	// cycle through coord system
	IF OptionsRtrig.Q AND NOT Controller.P_State.Buttons.Share THEN
		CASE _SMC_GroupJog2.CoordSystem OF
			SMC_COORD_SYSTEM.ACS:
				_SMC_GroupJog2.CoordSystem := SMC_COORD_SYSTEM.MCS;
				Controller.M_SetPlayerID(E_ControllerPlayerID.Player2);
			SMC_COORD_SYSTEM.MCS:
				_SMC_GroupJog2.CoordSystem := SMC_COORD_SYSTEM.PCS_1;
				Controller.M_SetPlayerID(E_ControllerPlayerID.Player3);
			SMC_COORD_SYSTEM.PCS_1:
				_SMC_GroupJog2.CoordSystem := SMC_COORD_SYSTEM.PCS_2;
				Controller.M_SetPlayerID(E_ControllerPlayerID.Player4);
			SMC_COORD_SYSTEM.PCS_2:
				_SMC_GroupJog2.CoordSystem := SMC_COORD_SYSTEM.TCS;
				Controller.M_SetPlayerID(E_ControllerPlayerID.PlayerALL);
			SMC_COORD_SYSTEM.TCS:
				_SMC_GroupJog2.CoordSystem := SMC_COORD_SYSTEM.ACS; // skip WCS
				Controller.M_SetPlayerID(E_ControllerPlayerID.Player1);
			SMC_COORD_SYSTEM.WCS:
				_SMC_GroupJog2.CoordSystem := SMC_COORD_SYSTEM.ACS;
				Controller.M_SetPlayerID(E_ControllerPlayerID.Player1);
		END_CASE
	END_IF
	
	// toggle the ABC as ACS setting
	IF ShareRtrig.Q AND NOT Controller.P_State.Buttons.Options THEN
		_SMC_GroupJog2.ABC_as_ACS := NOT _SMC_GroupJog2.ABC_as_ACS;
	END_IF
	
	// set the velocity factor while the left trigger button is pressed
	IF Controller.P_State.Dpad.Left AND_THEN Controller.P_State.Triggers.Right.Two <> R2_Last THEN
		R2_Last := Controller.P_State.Triggers.Right.Two;
		_SMC_GroupJog2.VelFactor := MAX(FactorMin, Controller.P_State.Triggers.Right.Two * 1.0 / 255.0);
	END_IF
	// set the acceleration factor while the up dpad button is pressed
	IF Controller.P_State.Dpad.Up AND_THEN Controller.P_State.Triggers.Right.Two <> R2_Last THEN
		R2_Last := Controller.P_State.Triggers.Right.Two;
		_SMC_GroupJog2.AccFactor := MAX(FactorMin, Controller.P_State.Triggers.Right.Two * 1.0 / 255.0);
	END_IF
	// set the jerk factor while the right dpad button is pressed
	IF Controller.P_State.Dpad.Right AND_THEN Controller.P_State.Triggers.Right.Two <> R2_Last THEN
		R2_Last := Controller.P_State.Triggers.Right.Two;
		_SMC_GroupJog2.JerkFactor := MAX(FactorMin, Controller.P_State.Triggers.Right.Two * 1.0 / 255.0);
	END_IF
	// set the torque factor while the down dpad down is pressed
	IF Controller.P_State.Dpad.Down AND_THEN Controller.P_State.Triggers.Right.Two <> R2_Last THEN
		R2_Last := Controller.P_State.Triggers.Right.Two;
		_SMC_GroupJog2.TorqueFactor := MAX(FactorMin, Controller.P_State.Triggers.Right.Two * 1.0 / 255.0);
	END_IF
	
	// first 4 poses can be called using buttons
	SquareButtonRtrig(CLK:=Controller.P_State.Buttons.Square);
	IF SquareButtonRtrig.Q THEN
		M_MoveToPose(E_Pose.One);
	END_IF
	TriangleButtonRtrig(CLK:=Controller.P_State.Buttons.Triangle);
	IF TriangleButtonRtrig.Q THEN
		M_MoveToPose(E_Pose.Two);
	END_IF
	CircleButtonRtrig(CLK:=Controller.P_State.Buttons.Circle);
	IF CircleButtonRtrig.Q THEN
		M_MoveToPose(E_Pose.Three);
	END_IF
	CrossButtonRtrig(CLK:=Controller.P_State.Buttons.Cross);
	IF CrossButtonRtrig.Q THEN
		M_MoveToPose(E_Pose.Four);
	END_IF
	
	//
	IF _SequenceMain = STEP_WAIT_JOG THEN
		
		//
		IF Controller.P_State.Joysticks.Left.X <> JoyStickLeftXLast
			OR Controller.P_State.Joysticks.Left.Y <> JoyStickLeftYLast THEN
				//
				JoyStickLeftXLast := Controller.P_State.Joysticks.Left.X;
				JoyStickLeftYLast := Controller.P_State.Joysticks.Left.Y;
				//	
				IF NOT Controller.P_State.Triggers.Left.One THEN
					// disable
					_SMC_GroupJog2.Forward[0] := FALSE;
					// disable
					_SMC_GroupJog2.Backward[0] := FALSE;
					// Controller.P_State.Joysticks.Left.X // X0-128 is -Y (Backward[1])
					_SMC_GroupJog2.Backward[1] := Controller.P_State.Joysticks.Left.X < _ControllerCenter - _ControllerDeadZone;
					// Controller.P_State.Joysticks.Left.X // X128-256 is +Y (Forward[1])
					_SMC_GroupJog2.Forward[1] := Controller.P_State.Joysticks.Left.X > _ControllerCenter + _ControllerDeadZone;
					// Controller.P_State.Joysticks.Left.Y // Y0-128 is +Z (Forward[2])
					_SMC_GroupJog2.Forward[2] := Controller.P_State.Joysticks.Left.Y < _ControllerCenter - _ControllerDeadZone;
					// Controller.P_State.Joysticks.Left.Y // Y128-256 is -Z (Backward[2])
					_SMC_GroupJog2.Backward[2] := Controller.P_State.Joysticks.Left.Y > _ControllerCenter + _ControllerDeadZone;
				ELSE
					// Controller.P_State.Joysticks.Left.Y // Y0-128 is +X (Forward[0])
					_SMC_GroupJog2.Forward[0] := Controller.P_State.Joysticks.Left.Y < _ControllerCenter - _ControllerDeadZone;
					// Controller.P_State.Joysticks.Left.Y // Y128-256 is -X (Backward[0])
					_SMC_GroupJog2.Backward[0] := Controller.P_State.Joysticks.Left.Y > _ControllerCenter + _ControllerDeadZone;
					// disable
					_SMC_GroupJog2.Backward[1] := FALSE;
					// disable
					_SMC_GroupJog2.Forward[1] := FALSE;
					// disable
					_SMC_GroupJog2.Forward[2] := FALSE;
					// disable])
					_SMC_GroupJog2.Backward[2] := FALSE;
				END_IF
		END_IF

		//
		IF Controller.P_State.Joysticks.Right.X <> JoyStickRightXLast
			OR Controller.P_State.Joysticks.Right.Y <> JoyStickRightYLast THEN
				//
				JoyStickRightXLast := Controller.P_State.Joysticks.Right.X;
				JoyStickRightYLast := Controller.P_State.Joysticks.Right.Y;
				//				
				IF NOT Controller.P_State.Triggers.Right.One THEN
					// Controller.P_State.Joysticks.Right.X // X0-128 is +Roll (rot about x) (Forward[3])
					_SMC_GroupJog2.Backward[3] := Controller.P_State.Joysticks.Right.X > _ControllerCenter + _ControllerDeadZone;
					// Controller.P_State.Joysticks.Right.X // X128-256 is -Roll (rot about x) (Backward[3])
					_SMC_GroupJog2.Forward[3] := Controller.P_State.Joysticks.Right.X < _ControllerCenter - _ControllerDeadZone;
					// Controller.P_State.Joysticks.Right.Y // Y0-128 is +Pitch (rot about y) (Forward[4])
					_SMC_GroupJog2.Forward[4] := Controller.P_State.Joysticks.Right.Y < _ControllerCenter - _ControllerDeadZone;
					// Controller.P_State.Joysticks.Right.Y // Y128-256 is -Pitch (rot about y) (Backward[4])
					_SMC_GroupJog2.Backward[4] := Controller.P_State.Joysticks.Right.Y > _ControllerCenter + _ControllerDeadZone;
					// disable
					_SMC_GroupJog2.Backward[5] := FALSE;
					// disable
					_SMC_GroupJog2.Forward[5] := FALSE;
				ELSE
					// disable
					_SMC_GroupJog2.Backward[3] := FALSE;
					// disable
					_SMC_GroupJog2.Forward[3] := FALSE;
					// disable
					_SMC_GroupJog2.Forward[4] := FALSE;
					// disable
					_SMC_GroupJog2.Backward[4] := FALSE;
					// Controller.P_State.Joysticks.Right.X // X0-128 is -Yaw (rot about z) (Backward[5])
					_SMC_GroupJog2.Backward[5] := Controller.P_State.Joysticks.Right.X < _ControllerCenter - _ControllerDeadZone;
					// Controller.P_State.Joysticks.Right.X // X128-256 is +Yaw (rot about z) (Forward[5])
					_SMC_GroupJog2.Forward[5] := Controller.P_State.Joysticks.Right.X > _ControllerCenter + _ControllerDeadZone;
				END_IF
		END_IF

	END_IF
	
END_IF
                        
END_METHOD

METHOD PRIVATE _M_CheckOffsets : BOOL
VAR_INPUT
END_VAR
VAR
	_i, _j, _k: INT;
END_VAR
                          IF _SMC_GroupJog2.Enable THEN
	FOR _j:=0 TO GVL.MCS_POS_IDX-GVL.TCP_POS_IDX BY 1 DO
		_OffsetExist[_j] := FALSE;
	END_FOR
	FOR _i := GVL.TCP_POS_IDX TO GVL.MCS_POS_IDX BY 1 DO
		IF StoredPositions[_i].Position.X <> 0
			OR_ELSE StoredPositions[_i].Position.Y <> 0
			OR_ELSE StoredPositions[_i].Position.Z <> 0
			OR_ELSE StoredPositions[_i].Position.A <> 0
			OR_ELSE StoredPositions[_i].Position.B <> 0
			OR_ELSE StoredPositions[_i].Position.C <> 0 THEN
				_OffsetExist[_i - GVL.TCP_POS_IDX] := TRUE;
		END_IF
	END_FOR
END_IF
                        
END_METHOD

METHOD PUBLIC M_ClearOffsets : BOOL
VAR_INPUT
END_VAR
                          
FOR _j:=0 TO 3 BY 1 DO
	_OffsetExist[_j] := FALSE;
END_FOR
FOR _i := GVL.TCP_POS_IDX TO GVL.MCS_POS_IDX BY 1 DO
	StoredPositions[_i].Position.X := 0.0;
	StoredPositions[_i].Position.Y := 0.0;
	StoredPositions[_i].Position.Z := 0.0;
	StoredPositions[_i].Position.A := 0.0;
	StoredPositions[_i].Position.B := 0.0;
	StoredPositions[_i].Position.C := 0.0;
END_FOR
                        
END_METHOD

METHOD PRIVATE _M_HandlePose : BOOL
VAR_IN_OUT
	AxisGroup: AXIS_GROUP_REF_SM3;
	GroupHandler: FB_GroupHandler;
END_VAR
VAR_INPUT
END_VAR
VAR
	_MoveCommand: ST_MoveCmd;
	_PoseSpeed: LREAL:=20.0;
END_VAR
                          FOR _i:=0 TO GVL.POSE_5_IDX - GVL.POSE_1_IDX BY 1 DO
	IF _MoveToPose[_i] THEN
		_MoveToPose[_i] := FALSE;
		//
		IF GVL.Enable 
			AND_THEN PersistentVars.Flags[GVL.HOME_COMPLETE].Value
			AND_THEN NOT _MoveCommandProcessor.Busy
			AND_THEN NOT _MoveCommandProcessor.Error THEN
				//
				_MoveCommand.MoveType 			:= DUT_Command_MoveType.DirectMove;
				_MoveCommand.PositionType 		:= DUT_Command_PositionType.AbsolutePosition;
				_MoveCommand.CoordinateType 	:= DUT_Command_CoordinateType.Literal;
				_MoveCommand.Speed 				:= _PoseSpeed;
				_MoveCommand.CoordSystem 		:= SMC_COORD_SYSTEM.ACS;
				_MoveCommand.CoordRef 			:= PersistentVars.StoredPositions[GVL.POSE_1_IDX + _i].Position;
				//
				_MoveCommandProcessor.Command := F_BuildMoveCmd(_MoveCommand);
				_MoveCommandProcessor.M_Start();
				//
				EXIT;
		END_IF;
	END_IF
END_FOR

_MoveCommandProcessor(
	StoredPositions:= StoredPositions,
	VisionRegisters:= VisionRegisters,
	Flags:= Flags,
	AxisGroup:= AxisGroup, 
	GroupHandler:= GroupHandler,
	Velocity:= StoredPositions[GVL.SPEEDS_IDX].Position.X, 
	VelFactor:= StoredPositions[GVL.SPEEDS_IDX].Position.A,
	Acceleration:= StoredPositions[GVL.SPEEDS_IDX].Position.Y, 
	AccFactor:= StoredPositions[GVL.SPEEDS_IDX].Position.B,
	Jerk:= StoredPositions[GVL.SPEEDS_IDX].Position.Z,
	JerkFactor:= StoredPositions[GVL.SPEEDS_IDX].Position.C, 
	Position=> ,
	ItfUnitMode=> , 
	Error=> );
                        
END_METHOD

METHOD PUBLIC M_MoveToPose : BOOL
VAR_INPUT
	Pose: E_Pose;
END_VAR
                          IF Enabled 
	AND NOT _MoveCommandProcessor.Busy
	AND NOT _MoveCommandProcessor.Error THEN
		M_MoveToPose := TRUE;
		_MoveToPose[Pose] := TRUE;
ELSE
	M_MoveToPose := FALSE;
END_IF
                        
END_METHOD
END_FUNCTION_BLOCK

FUNCTION_BLOCK FB_CommandProcessor EXTENDS FB_Module
VAR_IN_OUT
	J1, J2, J3, J4, J5, J6: AXIS_REF_SM3;
	AxisGroup: AXIS_GROUP_REF_SM3;
	GroupHandler: FB_GroupHandler;
	CmdIO: ST_LogicCmdIO;
	PrgProcessor: FB_ProgramProcessor;
END_VAR
VAR_INPUT
	Enable: BOOL;
END_VAR
VAR_OUTPUT
	ItfActiveProcessorUnitMode: PACK_ML.IUnitMode;
	ItfActiveModule: ItfModule;
	StatusText: STRING(255);
    GCodeLines: ARRAY[0..SMC_GCodeViewer.c_uiLines] OF STRING;
END_VAR
VAR
	_Commands: ARRAY [GVL.PROG_CMDS_ARR_BEG..GVL.PROG_CMDS_ARR_END] OF DUT_Command;
	_DummyUnitMode: PACK_ML.UnitMode;
	_UnitModeCurrentState: PACK_ML.State;
	_ActiveCommand: DUT_Command;
	_CurrentCmdIdx: UINT;
	_ProcessMoveCommand: FB_MoveCmdProcessor;
	_ProcessPauseCommand: FB_PauseCmdProcessor;
	//_ProcessInputCommand: InputCommandProcessor;
	_ProcessOutputCommand: FB_OutputCmdProcessor;
	_ProcessorDoneRtrig: R_TRIG;
    _ProcessVisionCommand: REFERENCE TO FB_VisionCmdProcessor; // keep vision in separate task
	_ProcessVarSetCommand: FB_VarSetCmdProcessor;
	_ProcessCncCommand: FB_CncCmdProcessor;
	_ProcessLogicCommand: FB_LogicCmdProcessor;
    _ErrorRtrig: ARRAY[0..7] OF R_TRIG;
	_FirstScan: BOOL:=TRUE;
END_VAR

VAR CONSTANT
	_STEP_DONE: 			INT := 1000;
	_STEP_IDLE: 			INT := 0000;
	_STEP_CMD:				INT := 0010;
	_STEP_WAIT:				INT := 0020;
	_STEP_ERR:              INT := 0030;
END_VAR

                    // keep this reference at the top in case we reference this somewhere else first
// hint: originally this was an issue because of the done and reset bits being referenced first
_ProcessVisionCommand REF= _40_Vision.ProcessVisionCommand;

//
SUPER^();

//
IF _FirstScan THEN
	// will exception if we don't set this on first scan
	_DummyUnitMode(sName := 'Active Processor', 
					eInitialState := PACK_ML.State.Idle,
					xActive := TRUE);
	ItfActiveProcessorUnitMode := _DummyUnitMode;
END_IF

// this is at best a hack and needs to be rethought out.
// we logically cant assign a process as the active unit mode 
// at start up so we use this dummy one
CASE _DummyUnitMode.CurrentState OF
	PACK_ML.State.Stopped,
	PACK_ML.State.Aborted,
	PACK_ML.State.Held,
	PACK_ML.State.Suspended,
	PACK_ML.State.Complete,
	PACK_ML.State.Idle:
		//
	PACK_ML.State.Resetting,
	PACK_ML.State.Starting,
	PACK_ML.State.Execute,
	PACK_ML.State.Suspending,
	PACK_ML.State.UnSuspending,
	PACK_ML.State.Holding,
	PACK_ML.State.UnHolding,
	PACK_ML.State.Completing,
	PACK_ML.State.Aborting,
	PACK_ML.State.Stopping,
	PACK_ML.State.Clearing:
		_DummyUnitMode.ActingStateCompleted();
END_CASE

// PackML state machine implementation
_UnitModeCurrentState := SUPER^._UnitMode.CurrentState;

//
_ErrorRtrig[0](CLK:=_ProcessMoveCommand.Error);
IF _ErrorRtrig[0].Q THEN
	SUPER^.M_Error(Description:=CONCAT('Move Error: ', _ProcessMoveCommand.ErrorDescription));
	StatusText:=SUPER^.ErrorDescription;
END_IF
_ErrorRtrig[1](CLK:=_ProcessPauseCommand.Error);
IF _ErrorRtrig[1].Q THEN
	SUPER^.M_Error(Description:=CONCAT('Pause Error: ', _ProcessPauseCommand.ErrorDescription));
	StatusText:=SUPER^.ErrorDescription;
END_IF
(*
_ErrorRtrig[2](CLK:=_ProcessInputCommand.Error);
IF _ErrorRtrig[2].Q THEN
	SUPER^._M_Error(Description:=CONCAT('Input Error: ', _ProcessInputCommand.ErrorDescription));
	StatusText:=SUPER^.ErrorDescription;
END_IF*)
_ErrorRtrig[3](CLK:=_ProcessOutputCommand.Error);
IF _ErrorRtrig[3].Q THEN
	SUPER^.M_Error(Description:=CONCAT('Output Error: ', _ProcessOutputCommand.ErrorDescription));
	StatusText:=SUPER^.ErrorDescription;
END_IF 
_ErrorRtrig[4](CLK:=_ProcessVisionCommand.Error);      
IF _ErrorRtrig[4].Q THEN
	SUPER^.M_Error(Description:=CONCAT('Vision Error: ', _ProcessVisionCommand.ErrorDescription));
	StatusText:=SUPER^.ErrorDescription;
END_IF
_ErrorRtrig[5](CLK:=_ProcessVarSetCommand.Error);
IF _ErrorRtrig[5].Q THEN
	SUPER^.M_Error(Description:=CONCAT('Variable Error: ', _ProcessVarSetCommand.ErrorDescription));
	StatusText:=SUPER^.ErrorDescription;
END_IF
_ErrorRtrig[6](CLK:=_ProcessCncCommand.Error);
IF _ErrorRtrig[6].Q THEN
	SUPER^.M_Error(Description:=CONCAT('CNC Error: ', _ProcessCncCommand.ErrorDescription));
	StatusText:=SUPER^.ErrorDescription;
END_IF
_ErrorRtrig[7](CLK:=_ProcessLogicCommand.Error);
IF _ErrorRtrig[7].Q THEN
	SUPER^.M_Error(Description:=CONCAT('Logic Error: ', _ProcessLogicCommand.ErrorDescription));
	StatusText:=SUPER^.ErrorDescription;
END_IF

_ProcessMoveCommand(
	StoredPositions:= SUPER^.StoredPositions,
	VisionRegisters:= SUPER^.VisionRegisters,
	Flags:= SUPER^.Flags,
	AxisGroup:= AxisGroup,
	GroupHandler:= GroupHandler,
	Velocity:= PersistentVars.StoredPositions[GVL.SPEEDS_IDX].Position.X, 
	VelFactor:= PersistentVars.StoredPositions[GVL.SPEEDS_IDX].Position.A,
	Acceleration:= PersistentVars.StoredPositions[GVL.SPEEDS_IDX].Position.Y, 
	AccFactor:= PersistentVars.StoredPositions[GVL.SPEEDS_IDX].Position.B,
	Jerk:= PersistentVars.StoredPositions[GVL.SPEEDS_IDX].Position.Z,
	JerkFactor:= PersistentVars.StoredPositions[GVL.SPEEDS_IDX].Position.C, 
	Position=> ,
	ItfUnitMode=>, 
	Error=> );

_ProcessPauseCommand(
	StoredPositions:= SUPER^.StoredPositions,
	VisionRegisters:= SUPER^.VisionRegisters,
	Flags:= SUPER^.Flags, 
	ElapsedTime=> , 
	RemainingTime=> , 
	ItfUnitMode=>, 
	Error=> );

//_ProcessInputCommand();
_ProcessOutputCommand(
	StoredPositions:= SUPER^.StoredPositions,
	VisionRegisters:= SUPER^.VisionRegisters,
	Flags:= SUPER^.Flags,
	Digital:= CmdIO.Output,
	Pwm:= CmdIO.Pwm,
	Enable:= Enable,
	ItfUnitMode=>, 
	Error=> );
	
_ProcessVarSetCommand( 
	StoredPositions:= SUPER^.StoredPositions,
	VisionRegisters:= SUPER^.VisionRegisters,
	Flags:= SUPER^.Flags,
	ItfUnitMode=>, 
	Error=> , 
	ErrorDescription=> );

_ProcessCncCommand(
	StoredPositions:= SUPER^.StoredPositions,
	VisionRegisters:= SUPER^.VisionRegisters,
	Flags:= SUPER^.Flags,
	J1:=J1, J2:=J2, J3:=J3, J4:=J4, J5:=J5, J6:=J6,
	AxisGroup:= AxisGroup, 
    CmdIO:= CmdIO,
    GCodeLines => GCodeLines,
	GapJerk:= , 
	GapVelocity:= , 
	AvoidGaps:= , 
	GapAccel:= , 
	ItfUnitMode=>, 
	Error=> , 
	ErrorDescription=> );
	
_ProcessLogicCommand(
	StoredPositions:= SUPER^.StoredPositions,
	VisionRegisters:= SUPER^.VisionRegisters,
	Flags:= SUPER^.Flags,
	CmdProcessor:= THIS^,
	PrgProcessor:= PrgProcessor,
	ItfUnitMode=>, 
	Error=> , 
	ErrorDescription=> , 
	CmdIO:= CmdIO);
	
_FirstScan := FALSE;
                  

METHOD PROTECTED M_Complete : BOOL
                          // once complete, reset to get back to idle
SUPER^._UnitMode.Reset();
                        
END_METHOD

METHOD PROTECTED M_Resetting : BOOL
                          CASE _SeqResetting OF
	0:
		_ProcessMoveCommand.M_Home();
		_ProcessPauseCommand.M_Home();
		//_ProcessInputCommand.M_Home();
		_ProcessOutputCommand.M_Home();
		_ProcessVisionCommand.M_Home();
		_ProcessVarSetCommand.M_Home();
		_ProcessCncCommand.M_Home();
		_ProcessLogicCommand.M_Home();
        StatusText := 'Resetting';
		_SeqResetting := _SeqResetting + 1;
	1:
		IF _ProcessMoveCommand.PropCurrentState = PACK_ML.State.Idle
			AND _ProcessPauseCommand.PropCurrentState = PACK_ML.State.Idle 
			//AND _ProcessInputCommand.PropCurrentState = PACK_ML.State.Idle
			AND _ProcessOutputCommand.PropCurrentState = PACK_ML.State.Idle
			AND _ProcessVisionCommand.PropCurrentState = PACK_ML.State.Idle
			AND _ProcessVarSetCommand.PropCurrentState = PACK_ML.State.Idle
			AND _ProcessCncCommand.PropCurrentState = PACK_ML.State.Idle
			AND _ProcessLogicCommand.PropCurrentState = PACK_ML.State.Idle THEN
				_SeqResetting := 0;
                StatusText := 'Idle';
				SUPER^.M_StateComplete();
		END_IF
		
END_CASE

SUPER^.M_Reset();

(*IF ItfActiveModule <> 0 THEN
	CASE _Seq OF
		0:
			IF NOT ItfActiveModule.PropCurrentState = PACK_ML.State.Idle THEN
				ItfActiveModule.M_Home();
				_Seq := 1;
			ELSE
				SUPER^.M_StateComplete();
			END_IF
		1:
			IF ItfActiveModule.PropCurrentState = PACK_ML.State.Idle THEN
				_Seq := 0;
			END_IF
			
	END_CASE
	
ELSE
	SUPER^.M_StateComplete();
	_Seq := 0;
	
END_IF*)
                        
END_METHOD

METHOD PUBLIC M_SetNextCommand : BOOL // returns true if successful
VAR_INPUT
	CommandNumber: UINT;
END_VAR
                          IF CommandNumber <= GVL.PROG_CMDS_ARR_END AND CommandNumber >= GVL.PROG_CMDS_ARR_BEG THEN
	_CurrentCmdIdx := CommandNumber;
	M_SetNextCommand := TRUE;
ELSE
	M_SetNextCommand := FALSE;
END_IF
                        
END_METHOD

METHOD PROTECTED M_Idle : BOOL
                          // in this state, we want to reset all the function blocks and hang out
_SeqMain := _STEP_IDLE;
_SeqAborting := 0;
_SeqClearing := 0;
_SeqResetting := 0;
                        
END_METHOD

METHOD PROTECTED M_SetPackML : BOOL
                          // SUPER already does this but the default is eInitialState:=PACK_ML.State.Idle 
// and we want PACK_ML.State.Aborted for the Orchestrator
SUPER^._UnitMode(sName := 'Command Processor',
				eInitialState := PACK_ML.State.Aborted,
				xActive := TRUE);
                        
END_METHOD

METHOD PROTECTED M_Starting : BOOL
                          // here we want to clear things and get ready for the execute state
// we can consider this the "INIT" state
_SeqMain := _STEP_CMD;
SUPER^._TimeoutTimer.PT := T#0MS; // timeout is ignored if set to 0
SUPER^.M_StateComplete();
                        
END_METHOD

METHOD PROTECTED M_Execute : BOOL
VAR
    _ErrorDescription: STRING;
END_VAR
                          // here we want to execute our commands/jobs/etc and set completed when done.
//
CASE _SeqMain OF
  	_STEP_DONE:
		_SeqMain := _STEP_IDLE;
		
	_STEP_IDLE:
		// hang out here until called to run
		_CurrentCmdIdx := 0;
		SUPER^.M_StateComplete();
		
	_STEP_CMD: //
		IF NOT Enable THEN
			_SeqMain := _STEP_DONE;
            _ErrorDescription := '';
            IF NOT GVL.Enable THEN
                _ErrorDescription := 'Robot not enabled';
            END_IF
            IF NOT PersistentVars.Flags[GVL.HOME_COMPLETE].Value THEN
                _ErrorDescription := CONCAT(_ErrorDescription, ' | Robot not homed');
            END_IF
            IF GVL.xActiveAlarm THEN
                _ErrorDescription := CONCAT(_ErrorDescription, ' | Active alarms exist');
            END_IF
            IF _ErrorDescription = '' THEN
                _ErrorDescription := 'Not enabled';
            END_IF
            _M_Error(Description := _ErrorDescription);
            
		ELSIF _CurrentCmdIdx <= GVL.PROG_CMDS_ARR_END AND _CurrentCmdIdx >= GVL.PROG_CMDS_ARR_BEG THEN
			//
			IF _Commands[_CurrentCmdIdx].CommandType = DUT_CommandType.Disabled THEN
				// want to increment here so that we can disable some commands 
				// in the program and it continue to execute
				_CurrentCmdIdx := _CurrentCmdIdx + 1;
				_SeqMain := _STEP_CMD;
				
			ELSE
				CASE _Commands[_CurrentCmdIdx].CommandType OF
					DUT_CommandType.MoveCommand: //
						StatusText := 'Move Command in Progress';
						ItfActiveProcessorUnitMode := _ProcessMoveCommand.ItfUnitMode;
						ItfActiveModule := _ProcessMoveCommand;
						_ProcessMoveCommand.Command := _Commands[_CurrentCmdIdx].CommandString;
						ItfActiveModule.M_Start();
					
					DUT_CommandType.PauseCommand: //
						StatusText := 'Pause Command in Progress';
						ItfActiveProcessorUnitMode := _ProcessPauseCommand.ItfUnitMode;
						ItfActiveModule := _ProcessPauseCommand;
						_ProcessPauseCommand.Command := _Commands[_CurrentCmdIdx].CommandString;
						ItfActiveModule.M_Start();
					
					DUT_CommandType.InputCommand: //
						StatusText := 'Input Command in Progress';
						//ActiveUnitMode := _ProcessInputCommand.ItfUnitMode;
						//ItfActiveModule := _ProcessInputCommand;
						//_ProcessInputCommand.Command := _Commands[_CurrentCmdIdx].CommandString;
						//ItfActiveModule.M_Start();
					
					DUT_CommandType.OutputCommand: //
						StatusText := 'Output Command in Progress';
						ItfActiveProcessorUnitMode := _ProcessOutputCommand.ItfUnitMode;
						ItfActiveModule := _ProcessOutputCommand;
						_ProcessOutputCommand.Command := _Commands[_CurrentCmdIdx].CommandString;
						ItfActiveModule.M_Start();
					
					DUT_CommandType.VisionCommand: //
						StatusText := 'Vision Command in Progress';
						ItfActiveProcessorUnitMode := _ProcessVisionCommand.ItfUnitMode;
						ItfActiveModule := _ProcessVisionCommand;
						_ProcessVisionCommand.Command := _Commands[_CurrentCmdIdx].CommandString;
						ItfActiveModule.M_Start();
					
					DUT_CommandType.VarSetCommand: //
						StatusText := 'VarSet Command in Progress';
						ItfActiveProcessorUnitMode := _ProcessVarsetCommand.ItfUnitMode;
						ItfActiveModule := _ProcessVarsetCommand;
						_ProcessVarsetCommand.Command := _Commands[_CurrentCmdIdx].CommandString;
						ItfActiveModule.M_Start();
					
					DUT_CommandType.CncCommand: //
						StatusText := 'CNC Command in Progress';
						ItfActiveProcessorUnitMode := _ProcessCncCommand.ItfUnitMode;
						ItfActiveModule := _ProcessCncCommand;
						_ProcessCncCommand.Command := _Commands[_CurrentCmdIdx].CommandString;
						ItfActiveModule.M_Start();
					
					DUT_CommandType.LogicCommand: //
						StatusText := 'Logic Command in Progress';
						ItfActiveProcessorUnitMode := _ProcessLogicCommand.ItfUnitMode;
						ItfActiveModule := _ProcessLogicCommand;
						_ProcessLogicCommand.Command := _Commands[_CurrentCmdIdx].CommandString;
						ItfActiveModule.M_Start();
						
				ELSE
					_SeqMain := _STEP_CMD;
					
				END_CASE
				
				// wait for executing
				IF ItfActiveModule.PropCurrentState = PACK_ML.State.Execute THEN
					_ActiveCommand := _Commands[_CurrentCmdIdx];
					_CurrentCmdIdx := _CurrentCmdIdx + 1;
					_SeqMain := _STEP_WAIT;
				END_IF
			END_IF
				
		ELSE
			_SeqMain := _STEP_DONE;
		END_IF
		
	_STEP_WAIT: // wait for command to finish
		//
		IF _ProcessorDoneRtrig.Q THEN
			_SeqMain := _STEP_CMD;
		END_IF
		//
		IF ItfActiveModule.PropError THEN
			SUPER^._UnitMode.Suspend();
			_SeqMain := _STEP_ERR;
		END_IF
		
	_STEP_ERR: //
	
END_CASE

// watch for rising edge of idle state. this was done for all processors since 
// the vision processor runs in a separate task and isnt guaranteed to start in the same 
// PLC scan.
_ProcessorDoneRtrig(clk:=ItfActiveProcessorUnitMode.CurrentState = PACK_ML.State.Idle);
                        
END_METHOD

METHOD PROTECTED M_Suspending : BOOL
                          IF ItfActiveModule <> 0 THEN
	IF ItfActiveModule.PropCurrentState = PACK_ML.State.Execute THEN
		ItfActiveModule.M_Hold();
		IF ItfActiveModule.PropCurrentState = PACK_ML.State.Held THEN
			SUPER^.M_StateComplete();
		END_IF
	ELSE
		SUPER^.M_StateComplete();
	END_IF
	
ELSE
	SUPER^.M_StateComplete();
	
END_IF
                        
END_METHOD

METHOD PROTECTED M_UnSuspending : BOOL
                          //
IF ItfActiveModule <> 0 THEN
	ItfActiveModule.M_Start();
	IF ItfActiveModule.PropCurrentState = PACK_ML.State.Execute THEN
		SUPER^.M_StateComplete();
	END_IF
	
ELSE
	SUPER^.M_StateComplete();
	
END_IF

//
_SeqMain := _STEP_WAIT;
                        
END_METHOD

METHOD PROTECTED M_Holding : BOOL
                          IF ItfActiveModule <> 0 THEN
	ItfActiveModule.M_Hold();
	IF ItfActiveModule.PropCurrentState = PACK_ML.State.Held THEN
		SUPER^.M_StateComplete();
	END_IF
ELSE
	SUPER^.M_StateComplete();
END_IF
                        
END_METHOD

METHOD PROTECTED M_Unholding : BOOL
                          //
IF ItfActiveModule <> 0 THEN
	ItfActiveModule.M_Start();
	IF ItfActiveModule.PropCurrentState = PACK_ML.State.Execute THEN
		SUPER^.M_StateComplete();
	END_IF
	
ELSE
	SUPER^.M_StateComplete();
	
END_IF

//
_SeqMain := _STEP_WAIT;
                        
END_METHOD

METHOD PROTECTED M_Aborting : BOOL
                          CASE _SeqAborting OF
	0:
		_ProcessMoveCommand.M_Abort();
		_ProcessPauseCommand.M_Abort();
		//_ProcessInputCommand.M_Abort();
		_ProcessOutputCommand.M_Abort();
		_ProcessVisionCommand.M_Abort();
		_ProcessVarSetCommand.M_Abort();
		_ProcessCncCommand.M_Abort();
		_ProcessLogicCommand.M_Abort();
		_SeqAborting := _SeqAborting + 1;
	1:
		IF _ProcessMoveCommand.PropCurrentState = PACK_ML.State.Aborted
			AND _ProcessPauseCommand.PropCurrentState = PACK_ML.State.Aborted 
			//AND _ProcessInputCommand.PropCurrentState = PACK_ML.State.Aborted
			AND _ProcessOutputCommand.PropCurrentState = PACK_ML.State.Aborted
			AND _ProcessVisionCommand.PropCurrentState = PACK_ML.State.Aborted
			AND _ProcessVarSetCommand.PropCurrentState = PACK_ML.State.Aborted
			AND _ProcessCncCommand.PropCurrentState = PACK_ML.State.Aborted
			AND _ProcessLogicCommand.PropCurrentState = PACK_ML.State.Aborted THEN
				_SeqAborting := 0;
				SUPER^.M_StateComplete();
		END_IF
		
END_CASE

(*IF ItfActiveModule <> 0 THEN
	ItfActiveModule.M_Abort();
	IF ItfActiveModule.PropCurrentState = PACK_ML.State.Aborted THEN
		SUPER^.M_StateComplete();
	END_IF
ELSE
	SUPER^.M_StateComplete();
END_IF*)
                        
END_METHOD

METHOD PROTECTED M_Stopping : BOOL
                          IF ItfActiveModule <> 0 THEN
	ItfActiveModule.M_Stop();
	IF ItfActiveModule.PropCurrentState = PACK_ML.State.Idle 
		OR ItfActiveModule.PropCurrentState = PACK_ML.State.Stopped 
		OR ItfActiveModule.PropCurrentState = PACK_ML.State.Aborted 
		OR ItfActiveModule.PropCurrentState = PACK_ML.State.Complete THEN
			SUPER^.M_StateComplete();
	END_IF
	
ELSE
	SUPER^.M_StateComplete();
	
END_IF
                        
END_METHOD

METHOD PROTECTED M_Clearing : BOOL
                          SUPER^.M_StateComplete();

(*IF SUPER^.Flags[GVL.HOME_COMPLETE].Value THEN
	CASE _SeqClearing OF
		0:
			_ProcessMoveCommand.M_Home();
			_SeqClearing := _SeqClearing + 1;
		1:
			IF _ProcessMoveCommand.PropCurrentState = PACK_ML.State.Idle THEN
				_SeqClearing := _SeqClearing + 1;
			END_IF
		2:
			IF NOT _ProcessMoveCommand.Error THEN
				_ProcessMoveCommand.Command := GVL.Pose2;
				_ProcessMoveCommand.M_Start();
				_SeqClearing := _SeqClearing + 1;
			ELSE
				SUPER^._M_Error(Description:='Move processor errored. Please reset and try again');
				_SeqClearing := -1;
			END_IF
		3:
			IF _ProcessMoveCommand.PropCurrentState = PACK_ML.State.Execute THEN
				_SeqClearing := _SeqClearing + 1;
			END_IF
		4:
			IF _ProcessMoveCommand.PropCurrentState = PACK_ML.State.Complete 
				OR _ProcessMoveCommand.PropCurrentState = PACK_ML.State.Stopped 
				OR _ProcessMoveCommand.PropCurrentState = PACK_ML.State.Aborted
				OR _ProcessMoveCommand.PropCurrentState = PACK_ML.State.Idle  THEN
					SUPER^.M_StateComplete();
					_SeqClearing := 0;
			END_IF
	END_CASE
ELSE
	SUPER^._M_Error(Description:='Drives are not homed. Please home and try again');
	_SeqClearing := -1;
END_IF

IF _ProcessMoveCommand.Error THEN
	SUPER^._M_Error(Description:='Move processor in error state. Please reset and try again');
	_SeqClearing := -1;
END_IF
*)

(*
IF ItfActiveModule <> 0 THEN
	//
	CASE _Seq OF
		0:
			IF NOT ItfActiveModule.PropCurrentState = PACK_ML.State.Stopped THEN
				ItfActiveModule.M_Abort();
				_Seq := 1;
			ELSE
				SUPER^.M_StateComplete();
			END_IF
		1:
			CASE ItfActiveModule.PropCurrentState OF
				PACK_ML.State.Aborted:
					ItfActiveModule.Clear();
				PACK_ML.State.Stopped:
					_Seq := 0;
			END_CASE
			
	END_CASE
ELSE
	_Seq := 0;
	SUPER^.M_StateComplete();
END_IF
*)

                        
END_METHOD

METHOD PUBLIC M_SetCommands : BOOL
VAR_INPUT
	StartingCommand: UINT;
	Commands: ARRAY [GVL.PROG_CMDS_ARR_BEG..GVL.PROG_CMDS_ARR_END] OF DUT_Command;
END_VAR
                          IF StartingCommand >= GVL.PROG_CMDS_ARR_BEG AND StartingCommand <= GVL.PROG_CMDS_ARR_END + 1 THEN // +1 because we want to be able to tell if calling program was on last command
	_CurrentCmdIdx := StartingCommand;
	_Commands := Commands;
	M_SetCommands := TRUE;
ELSE
	M_SetCommands := FALSE;
END_IF
                        
END_METHOD

METHOD PRIVATE _M_Error
VAR_INPUT
    Description: STRING;
END_VAR
                          SUPER^.M_Error(Description := CONCAT('Command Processor: ', Description));
                        
END_METHOD

{attribute 'monitoring' := 'variable'}
PROPERTY PUBLIC P_CurrentCommandIndex : REFERENCE TO UINT
GET
VAR
END_VAR
                            P_CurrentCommandIndex REF= _CurrentCmdIdx;
                          
END_GET
END_PROPERTY

{attribute 'monitoring' := 'variable'}
PROPERTY PUBLIC P_CurrentCommand : REFERENCE TO DUT_Command
GET
VAR
END_VAR
                            P_CurrentCommand REF= _ActiveCommand;
                          
END_GET
END_PROPERTY
END_FUNCTION_BLOCK

FUNCTION_BLOCK FB_ParseMoveCmd
VAR_INPUT
	Command: STRING(GVL.COMMAND_LEN);
END_VAR
VAR_OUTPUT
	stCommand: ST_MoveCmd;
	Error: BOOL:= FALSE;
	ErrorDescription: STRING:='';
END_VAR
VAR
	_CmdParams: ARRAY [0..GVL.COMMAND_LEN] OF STRING;
END_VAR
VAR CONSTANT
	_MoveTypeD: STRING(3):='DIR';
	_MoveTypeL: STRING(3):='LIN';
	_MoveTypeC: STRING(3):='CIR';
	_ChangeTypeA: STRING(3):='ABS';
	_ChangeTypeR: STRING(3):='REL';
	_CoordSystemAcs: STRING(3):='ACS';
	_CoordSystemMcs: STRING(3):='MCS';
	_CoordSystemPc1: STRING(3):='PC1';
	_CoordSystemPc2: STRING(3):='PC2';
	_CoordSystemTcs: STRING(3):='TCS';
	_CoordSystemWcs: STRING(3):='WCS';
	_CoordSystemIcs: STRING(3):='ICS';
	_CoordTypeH: STRING(3):='LIT';
	_CoordTypeV: STRING(3):='VAR';
	_ArrayTypeS: STRING(3):='STO';
	_ArrayTypeV: STRING(3):='VIS';
	_ArrayTypeF: STRING(3):='FLG';
	_CircleModeBor: STRING(3):='BOR';
	_CircleModeCen: STRING(3):='CEN';
	_CircleModeRad: STRING(3):='RAD';
	_PathChoiceClw: STRING(3):='CLW';
	_PathChoiceCcw: STRING(3):='CCW';
END_VAR

                    // D is direct move. L is linear move. C is a circular move
// R is relative position. A is absolute position
// V is variable coordinated. H is a hardcoded coordinated
// S is stored position array. V is vision register array.
// D|L|C R|A Speed CoordSystem X0000.00 Y0000.00 Z0000.00 A0000.00 B0000.00 C0000.00 BOR|CEN|RAD CCW|CLW X0000.00 Y0000.00 Z0000.00 A0000.00 B0000.00 C0000.00
// 'D A 10 MCS H +0250.00 +0000.00 +0500.00 +0000.00 +0045.00 +0180.00'
// 'C R 10 MCS H +0250.00 +0000.00 +0500.00 +0000.00 +0045.00 +0180.00 BOR CLW H +0250.00 +0000.00 +0500.00 +0000.00 +0045.00 +0180.00'
// 'D A 10 MCS V S 25'
// 'D A 10 MCS V V 33'
// 'C R 10 MCS V S 2 BOR CLW V S 005'
// 'C R 10 MCS V S 003 BOR CLW V V 006'
// 'C R 10 MCS V S 015 BOR CLW H +0250.00 +0000.00 +0500.00 +0000.00 +0045.00 +0180.00'
// 'C R 10 MCS H 250.0 0.0 500.0 0.0 45.0 180.0 BOR CLW V V 22'

Error := FALSE;
ErrorDescription := '';

// split command string into commands
_CmdParams:=F_SplitCmd(Command:=Command);

//
IF _CmdParams[0] = _MoveTypeD THEN
	stCommand.MoveType := DUT_Command_MoveType.DirectMove;
ELSIF _CmdParams[0] = _MoveTypeL THEN
	stCommand.MoveType := DUT_Command_MoveType.LinearMove;
ELSIF _CmdParams[0] = _MoveTypeC THEN
	stCommand.MoveType := DUT_Command_MoveType.CircularMove;
ELSE
	Error := TRUE;
	ErrorDescription := 'Incorrect move type';
END_IF

//
IF _CmdParams[1] = _ChangeTypeR THEN
	stCommand.PositionType := DUT_Command_PositionType.RelativePosition;
ELSIF _CmdParams[1] = _ChangeTypeA THEN
	stCommand.PositionType := DUT_Command_PositionType.AbsolutePosition;
ELSE
	Error := TRUE;
	ErrorDescription := 'Incorrect position type';
END_IF

//
stCommand.Speed := STRING_TO_LREAL(_CmdParams[2]);

//
IF _CmdParams[3] = _CoordSystemAcs THEN
	stCommand.CoordSystem := SMC_COORD_SYSTEM.ACS;
ELSIF _CmdParams[3] = _CoordSystemMcs THEN
	stCommand.CoordSystem := SMC_COORD_SYSTEM.MCS;
ELSIF _CmdParams[3] = _CoordSystemPc1 THEN
	stCommand.CoordSystem := SMC_COORD_SYSTEM.PCS_1;
ELSIF _CmdParams[3] = _CoordSystemPc2 THEN
	stCommand.CoordSystem := SMC_COORD_SYSTEM.PCS_2;
ELSIF _CmdParams[3] = _CoordSystemTcs THEN
	stCommand.CoordSystem := SMC_COORD_SYSTEM.TCS;
ELSIF _CmdParams[3] = _CoordSystemWcs THEN
	stCommand.CoordSystem := SMC_COORD_SYSTEM.WCS;
ELSIF _CmdParams[3] = _CoordSystemIcs THEN
	stCommand.CoordSystem := SMC_COORD_SYSTEM.ICS;
ELSE
	Error := TRUE;
	ErrorDescription := 'Incorrect coordinate system type';
END_IF

//
IF _CmdParams[4] = _CoordTypeH THEN
	stCommand.CoordinateType := DUT_Command_CoordinateType.Literal;
ELSIF _CmdParams[4] = _CoordTypeV THEN
	stCommand.CoordinateType := DUT_Command_CoordinateType.Variable;
ELSE
	Error := TRUE;
	ErrorDescription := 'Incorrect coordinate type'; // TODO wow i need a better name for this... wtf was i thinking?
END_IF

//
CASE stCommand.CoordinateType OF 
// 'D A 010 MCS H +0250.00 +0000.00 +0500.00 +0000.00 +0045.00 +0180.00'
	DUT_Command_CoordinateType.Literal:
		stCommand.CoordRef.X := STRING_TO_LREAL(_CmdParams[5]);
		stCommand.CoordRef.Y := STRING_TO_LREAL(_CmdParams[6]);
		stCommand.CoordRef.Z := STRING_TO_LREAL(_CmdParams[7]);
		stCommand.CoordRef.A := STRING_TO_LREAL(_CmdParams[8]);
		stCommand.CoordRef.B := STRING_TO_LREAL(_CmdParams[9]);
		stCommand.CoordRef.C := STRING_TO_LREAL(_CmdParams[10]);
// 'D A 010 MCS V S 001'
	DUT_Command_CoordinateType.Variable:
		stCommand.ArrayIndex := STRING_TO_UINT(_CmdParams[6]);
		IF stCommand.ArrayIndex <= GVL.POS_ARR_END 
			AND stCommand.ArrayIndex >= GVL.POS_ARR_BEG THEN
				IF _CmdParams[5] = _ArrayTypeS THEN
					stCommand.ArrayType := DUT_Command_ArrayType.StoredPosition;
					stCommand.CoordRef := PersistentVars.StoredPositions[stCommand.ArrayIndex].Position;
				ELSIF _CmdParams[5] = _ArrayTypeV THEN
					stCommand.ArrayType := DUT_Command_ArrayType.VisionRegister;
					stCommand.CoordRef := PersistentVars.VisionRegisters[stCommand.ArrayIndex].Position;
				ELSE
					Error := TRUE;
					ErrorDescription := 'Incorrect array type';
				END_IF
		ELSE
			Error := TRUE;
			ErrorDescription := 'Array index out of bounds';
		END_IF
	
END_CASE

//
CASE stCommand.CoordinateType OF 
// 'C R 010 MCS H +0250.00 +0000.00 +0500.00 +0000.00 +0045.00 +0180.00 BOR CLW H +0250.00 +0000.00 +0500.00 +0000.00 +0045.00 +0180.00'
	DUT_Command_CoordinateType.Literal:
		IF _CmdParams[11] = _CircleModeBor THEN
			stCommand.CircleMode := SMC_CIRC_MODE.BORDER;
		ELSIF _CmdParams[11] = _CircleModeCen THEN
			stCommand.CircleMode := SMC_CIRC_MODE.CENTER;
		ELSIF _CmdParams[11] = _CircleModeRad THEN
			stCommand.CircleMode := SMC_CIRC_MODE.RADIUS;
		ELSE
			Error := TRUE;
			ErrorDescription := 'Incorrect circle mode';
		END_IF
// 'C R 010 MCS V S 001 BOR CLW H +0250.00 +0000.00 +0500.00 +0000.00 +0045.00 +0180.00'
	DUT_Command_CoordinateType.Variable:
		IF _CmdParams[7] = _CircleModeBor THEN
			stCommand.CircleMode := SMC_CIRC_MODE.BORDER;
		ELSIF _CmdParams[7] = _CircleModeCen THEN
			stCommand.CircleMode := SMC_CIRC_MODE.CENTER;
		ELSIF _CmdParams[7] = _CircleModeRad THEN
			stCommand.CircleMode := SMC_CIRC_MODE.RADIUS;
		ELSE
			Error := TRUE;
			ErrorDescription := 'Incorrect circle mode';
		END_IF
	
END_CASE

//
CASE stCommand.CoordinateType OF 
// 'C R 010 MCS H +0250.00 +0000.00 +0500.00 +0000.00 +0045.00 +0180.00 BOR CLW H +0250.00 +0000.00 +0500.00 +0000.00 +0045.00 +0180.00'
	DUT_Command_CoordinateType.Literal:
		IF _CmdParams[12] = _PathChoiceClw THEN
			stCommand.PathChoice := MC_CIRC_PATHCHOICE.CLOCKWISE;
		ELSIF _CmdParams[12] = _PathChoiceCcw THEN
			stCommand.PathChoice := MC_CIRC_PATHCHOICE.COUNTER_CLOCKWISE;
		ELSE
			Error := TRUE;
			ErrorDescription := 'Incorrect circle direction';
		END_IF
		IF _CmdParams[13] = _CoordTypeH THEN
			stCommand.CircularCoordinateType := DUT_Command_CoordinateType.Literal;
		ELSIF _CmdParams[13] = _CoordTypeV THEN
			stCommand.CircularCoordinateType := DUT_Command_CoordinateType.Variable;
		ELSE
			Error := TRUE;
			ErrorDescription := 'Incorrect coordinate type'; // TODO yeah, this needs better naming. "coordinate type" does not fit.
		END_IF
// 'C R 010 MCS V S 001 BOR CLW H +0250.00 +0000.00 +0500.00 +0000.00 +0045.00 +0180.00'
	DUT_Command_CoordinateType.Variable:
		IF _CmdParams[8] = _PathChoiceClw THEN
			stCommand.PathChoice := MC_CIRC_PATHCHOICE.CLOCKWISE;
		ELSIF _CmdParams[8] = _PathChoiceCcw THEN
			stCommand.PathChoice := MC_CIRC_PATHCHOICE.COUNTER_CLOCKWISE;
		ELSE
			Error := TRUE;
			ErrorDescription := 'Incorrect circle direction';
		END_IF
		IF _CmdParams[9] = _CoordTypeH THEN
			stCommand.CircularCoordinateType := DUT_Command_CoordinateType.Literal;
		ELSIF _CmdParams[9] = _CoordTypeV THEN
			stCommand.CircularCoordinateType := DUT_Command_CoordinateType.Variable;
		ELSE
			Error := TRUE;
			ErrorDescription := 'Incorrect coordinate type'; // TODO this naming "coordinate type" needs to go.
		END_IF
	
END_CASE

//
CASE stCommand.CircularCoordinateType OF 
	DUT_Command_CoordinateType.Literal:
		CASE stCommand.CoordinateType OF
// 'C R 010 MCS H +0250.00 +0000.00 +0500.00 +0000.00 +0045.00 +0180.00 BOR CLW H +0250.00 +0000.00 +0500.00 +0000.00 +0045.00 +0180.00'
			DUT_Command_CoordinateType.Literal:
				stCommand.CoordRef2.X := STRING_TO_LREAL(_CmdParams[14]);
				stCommand.CoordRef2.Y := STRING_TO_LREAL(_CmdParams[15]);
				stCommand.CoordRef2.Z := STRING_TO_LREAL(_CmdParams[16]);
				stCommand.CoordRef2.A := STRING_TO_LREAL(_CmdParams[17]);
				stCommand.CoordRef2.B := STRING_TO_LREAL(_CmdParams[18]);
				stCommand.CoordRef2.C := STRING_TO_LREAL(_CmdParams[19]);
// 'C R 010 MCS V S 001 BOR CLW H +0250.00 +0000.00 +0500.00 +0000.00 +0045.00 +0180.00'
			DUT_Command_CoordinateType.Variable:
				stCommand.CoordRef2.X := STRING_TO_LREAL(_CmdParams[10]);
				stCommand.CoordRef2.Y := STRING_TO_LREAL(_CmdParams[11]);
				stCommand.CoordRef2.Z := STRING_TO_LREAL(_CmdParams[12]);
				stCommand.CoordRef2.A := STRING_TO_LREAL(_CmdParams[13]);
				stCommand.CoordRef2.B := STRING_TO_LREAL(_CmdParams[14]);
				stCommand.CoordRef2.C := STRING_TO_LREAL(_CmdParams[15]);
				
		END_CASE
	
	DUT_Command_CoordinateType.Variable:
		CASE stCommand.CoordinateType OF
// 'C R 010 MCS H +0250.00 +0000.00 +0500.00 +0000.00 +0045.00 +0180.00 BOR CLW V V 001'
			DUT_Command_CoordinateType.Literal:
				stCommand.CircularArrayIndex := STRING_TO_UINT(_CmdParams[15]);
				IF stCommand.CircularArrayIndex <= GVL.POS_ARR_END 
					AND stCommand.CircularArrayIndex >= GVL.POS_ARR_BEG THEN
						IF _CmdParams[14] = _ArrayTypeS THEN
							stCommand.CircularArrayType := DUT_Command_ArrayType.StoredPosition;
							stCommand.CoordRef2 := PersistentVars.StoredPositions[stCommand.CircularArrayIndex].Position;
						ELSIF _CmdParams[14] = _ArrayTypeV THEN
							stCommand.CircularArrayType := DUT_Command_ArrayType.VisionRegister;
							stCommand.CoordRef2 := PersistentVars.VisionRegisters[stCommand.CircularArrayIndex].Position;
						ELSE
							Error := TRUE;
							ErrorDescription := 'Incorrect array type';
						END_IF
					
				ELSE
					Error:=TRUE;
					ErrorDescription := 'Array index out of bounds';
					
				END_IF
				
// 'C R 010 MCS V S 001 BOR CLW V V 001'
			DUT_Command_CoordinateType.Variable:
				stCommand.CircularArrayIndex := STRING_TO_UINT(_CmdParams[11]);
				IF stCommand.CircularArrayIndex <= GVL.POS_ARR_END 
					AND stCommand.CircularArrayIndex >= GVL.POS_ARR_BEG THEN
						IF _CmdParams[10] = _ArrayTypeS THEN
							stCommand.CircularArrayType := DUT_Command_ArrayType.StoredPosition;
							stCommand.CoordRef2 := PersistentVars.StoredPositions[stCommand.CircularArrayIndex].Position;
						ELSIF _CmdParams[10] = _ArrayTypeV THEN
							stCommand.CircularArrayType := DUT_Command_ArrayType.VisionRegister;
							stCommand.CoordRef2 := PersistentVars.VisionRegisters[stCommand.CircularArrayIndex].Position;
						ELSE
							Error:=TRUE;
							ErrorDescription := 'Incorrect array type';
						END_IF
					
				ELSE
					Error:=TRUE;
					ErrorDescription := 'Array index out of bounds';
				END_IF
				
		END_CASE
	
END_CASE
                  
END_FUNCTION_BLOCK

PROGRAM _30_Visu
VAR	
    // alarms
	itfAlarmConfiguration : AlarmManager.IAlarmConfiguration;
    itfAlarmConfiguration7 : AlarmManager.IAlarmConfiguration7;
    iAlarmCfg : INT;
    
    //
	SelectedProgramNumber: INT;
	SelectedRecipeRowIndex: INT;
    SelectedRecipeRowIndexLast: INT;
	RecipeRowSelected: BOOL;
	InsertLineAbove: BOOL;
	InsertLineBelow: BOOL;
	DeleteLine: BOOL;
	CopySelectedCommand: BOOL;
	CopiedCommandType: DUT_CommandType;
	CopiedCommandString: STRING(GVL.COMMAND_LEN);
	CopiedCommandComment: STRING;
	PasteCommand: BOOL;
	JumpRowChanged: BOOL;
    ScrollingBegin: BOOL;
    ScrollingSingleUp: BOOL;
    ScrollingSingleDown: BOOL;
    ScrollingPageUp: BOOL;
    ScrollingPageDown: BOOL;
    ScrollingEnd: BOOL;
	
	_i,_j,_k: INT;
	
	SetStoredPositionAsCurrent: BOOL;
	SelectedStoredPosition: UINT;
	SetVisionRegisterAsCurrent: BOOL;
	SelectedVisionRegister: UINT;
	SelectedFlag: UINT;
	
	//
	TeachPosition: BOOL;
	stTeachPosition: ST_MoveCmd;
	
	//
	MoveCmdParser: FB_ParseMoveCmd;
	stMoveCmd: ST_MoveCmd;
	MoveCmdVisu: AddMoveCmd_VISU_STRUCT;
	
	//
	OutputCmdParser: FB_ParseOutputCmd;
	stOutputCmd: ST_OutputCmd;
	OutputCmdVisu: AddOutputCmd_VISU_STRUCT;
	
	//
	PauseCmdParser: FB_ParsePauseCmd;
	stPauseCmd: ST_PauseCmd;
	PauseCmdVisu: AddPauseCmd_VISU_STRUCT;
	
	//
	VisionCmdParser : FB_ParseVisionCmd;
	stVisionCmd : ST_VisionCmd;
	VisionCmdVisu: AddVisionCmd_VISU_STRUCT;
	
	//
	VarSetCmdParser : FB_ParseVarSetCmd;
	stVarSetCmd : ST_VarSetCmd;
	VarSetCmdVisu: AddVarSetCmd_VISU_STRUCT;
	
	//
	CncCmdParser : FB_ParseCncCmd;
	stCncCmd : ST_CncCmd;
	CncCmdVisu: AddCncCmd_VISU_STRUCT;
	
	//
	LogicCmdParser : FB_ParseLogicCmd;
	stLogicCmd : ST_LogicCmd;
	LogicCmdVisu: AddLogicCmd_VISU_STRUCT;
	
	//
	CurrentVisu: STRING;
	OpenDialog: VU.FbOpenDialogExtended;

END_VAR

                    //
GVL.lrGripperOpen := SEL(GVL.CmdIO.Output[0], 0.0, 100.0);

// scrolling
IF ScrollingBegin OR ScrollingSingleUp OR ScrollingSingleDown OR ScrollingPageUp OR ScrollingPageDown OR ScrollingEnd
    AND_THEN SelectedRecipeRowIndex <> SelectedRecipeRowIndexLast THEN
        SelectedRecipeRowIndexLast := SelectedRecipeRowIndex;
        ScrollingBegin := ScrollingSingleUp := ScrollingSingleDown := ScrollingPageUp := ScrollingPageDown := ScrollingEnd := FALSE;
END_IF

//
IF (InsertLineAbove OR InsertLineBelow) AND RecipeRowSelected THEN
	//
	IF InsertLineAbove THEN
		InsertLineAbove := FALSE;
		_j := SelectedRecipeRowIndex + 1;
	ELSIF InsertLineBelow THEN
		InsertLineBelow := FALSE;
		_j := SelectedRecipeRowIndex + 2;
	END_IF
	//
	FOR _i := GVL.PROG_CMDS_ARR_END TO _j BY -1 DO
		// shift all data
		IF _i >= GVL.PROG_CMDS_ARR_BEG AND _i <= GVL.PROG_CMDS_ARR_END THEN // can never really be too careful am I right?
			//
			MemUtils.MemCpy(pbyDest:=ADR(PersistentVars.Programs[SelectedProgramNumber].Commands[_i]),
							pbySrc:=ADR(PersistentVars.Programs[SelectedProgramNumber].Commands[_i - 1]),
							dwSize:=SIZEOF(PersistentVars.Programs[SelectedProgramNumber].Commands[_i]));
		END_IF
	END_FOR
	FOR _k := GVL.PROG_CMDS_ARR_END TO GVL.PROG_CMDS_ARR_BEG BY -1 DO
		// check if the command is a logic command with a jump function
		// if so, we need to move the jump row automatically so it doesnt point to an invalid command.
		// otherwise, the user would have to manually change this each time they move rows.
		JumpRowChanged := F_ChangeJumpRow(Command:=PersistentVars.Programs[SelectedProgramNumber].Commands[_k], BeginningRow:= _j-1, Change:= 1);
	END_FOR
	//
	PersistentVars.Programs[SelectedProgramNumber].Commands[_j - 1].CommandType := DUT_CommandType.Disabled;
	PersistentVars.Programs[SelectedProgramNumber].Commands[_j - 1].CommandString := '';
	PersistentVars.Programs[SelectedProgramNumber].Commands[_j - 1].CommandComment := '';
END_IF

//
IF DeleteLine AND RecipeRowSelected THEN
	DeleteLine := FALSE;
	FOR _i := SelectedRecipeRowIndex TO GVL.PROG_CMDS_ARR_END - 1 BY 1 DO
		IF _i >= GVL.PROG_CMDS_ARR_BEG AND _i <= GVL.PROG_CMDS_ARR_END THEN // can never really be too careful am I right?
			//
			MemUtils.MemCpy(pbyDest:=ADR(PersistentVars.Programs[SelectedProgramNumber].Commands[_i]),
							pbySrc:=ADR(PersistentVars.Programs[SelectedProgramNumber].Commands[_i + 1]),
							dwSize:=SIZEOF(PersistentVars.Programs[SelectedProgramNumber].Commands[_i]));
		END_IF
	END_FOR
	FOR _k := GVL.PROG_CMDS_ARR_END TO GVL.PROG_CMDS_ARR_BEG BY -1 DO
		// check if the command is a logic command with a jump function
		// if so, we need to move the jump row automatically so it doesnt point to an invalid command.
		// otherwise, the user would have to manually change this each time they move rows.
		JumpRowChanged := F_ChangeJumpRow(Command:=PersistentVars.Programs[SelectedProgramNumber].Commands[_k], BeginningRow:= SelectedRecipeRowIndex, Change:= -1);
	END_FOR
END_IF

//
IF SetStoredPositionAsCurrent THEN
	SetStoredPositionAsCurrent := FALSE;
	PersistentVars.StoredPositions[SelectedStoredPosition].Position.X := F_RoundLreal(_00_Main.ProcessJog.Position.v[0],2);
	PersistentVars.StoredPositions[SelectedStoredPosition].Position.Y := F_RoundLreal(_00_Main.ProcessJog.Position.v[1],2);
	PersistentVars.StoredPositions[SelectedStoredPosition].Position.Z := F_RoundLreal(_00_Main.ProcessJog.Position.v[2],2);
	PersistentVars.StoredPositions[SelectedStoredPosition].Position.A := F_RoundLreal(_00_Main.ProcessJog.Position.v[3],2);
	PersistentVars.StoredPositions[SelectedStoredPosition].Position.B := F_RoundLreal(_00_Main.ProcessJog.Position.v[4],2);
	PersistentVars.StoredPositions[SelectedStoredPosition].Position.C := F_RoundLreal(_00_Main.ProcessJog.Position.v[5],2);
END_IF

//
IF TeachPosition THEN
	TeachPosition := FALSE;
	//
	stTeachPosition.MoveType := DUT_Command_MoveType.DirectMove;
	stTeachPosition.Speed := 50;
	stTeachPosition.PositionType := DUT_Command_PositionType.AbsolutePosition;
	stTeachPosition.CoordSystem := _00_Main.ProcessJog.CoordSystem;
	stTeachPosition.CoordRef.X := F_RoundLreal(_00_Main.ProcessJog.Position.v[0],2);
	stTeachPosition.CoordRef.Y := F_RoundLreal(_00_Main.ProcessJog.Position.v[1],2);
	stTeachPosition.CoordRef.Z := F_RoundLreal(_00_Main.ProcessJog.Position.v[2],2);
	stTeachPosition.CoordRef.A := F_RoundLreal(_00_Main.ProcessJog.Position.v[3],2);
	stTeachPosition.CoordRef.B := F_RoundLreal(_00_Main.ProcessJog.Position.v[4],2);
	stTeachPosition.CoordRef.C := F_RoundLreal(_00_Main.ProcessJog.Position.v[5],2);
	PersistentVars.Programs[SelectedProgramNumber].Commands[SelectedRecipeRowIndex].CommandType := DUT_CommandType.MoveCommand;
	PersistentVars.Programs[SelectedProgramNumber].Commands[SelectedRecipeRowIndex].CommandString := F_BuildMoveCmd(stTeachPosition);
	PersistentVars.Programs[SelectedProgramNumber].Commands[SelectedRecipeRowIndex].CommandComment := 'Taught position';
END_IF

//
IF PasteCommand THEN
	PasteCommand := FALSE;
	PersistentVars.Programs[SelectedProgramNumber].Commands[SelectedRecipeRowIndex].CommandType := CopiedCommandType;
	PersistentVars.Programs[SelectedProgramNumber].Commands[SelectedRecipeRowIndex].CommandString := CopiedCommandString;
	PersistentVars.Programs[SelectedProgramNumber].Commands[SelectedRecipeRowIndex].CommandComment := CopiedCommandComment;
END_IF

//
IF CopySelectedCommand THEN
	CopySelectedCommand := FALSE;
	
	//
	CopiedCommandType := PersistentVars.Programs[SelectedProgramNumber].Commands[SelectedRecipeRowIndex].CommandType;
	CopiedCommandString := PersistentVars.Programs[SelectedProgramNumber].Commands[SelectedRecipeRowIndex].CommandString;
	CopiedCommandComment := PersistentVars.Programs[SelectedProgramNumber].Commands[SelectedRecipeRowIndex].CommandComment;
	
	CASE PersistentVars.Programs[SelectedProgramNumber].Commands[SelectedRecipeRowIndex].CommandType OF
		DUT_CommandType.Disabled:
			//
			
		DUT_CommandType.MoveCommand:
			MoveCmdParser(Command := PersistentVars.Programs[SelectedProgramNumber].Commands[SelectedRecipeRowIndex].CommandString);
			stMoveCmd := MoveCmdParser.stCommand;
			
		DUT_CommandType.PauseCommand:
			PauseCmdParser(Command:=PersistentVars.Programs[SelectedProgramNumber].Commands[SelectedRecipeRowIndex].CommandString);
			stPauseCmd := PauseCmdParser.stCommand;
			
		DUT_CommandType.InputCommand:
			//
			
		DUT_CommandType.OutputCommand:
			OutputCmdParser(Command:=PersistentVars.Programs[SelectedProgramNumber].Commands[SelectedRecipeRowIndex].CommandString);
			stOutputCmd := OutputCmdParser.stCommand;
			
		DUT_CommandType.VisionCommand:
			VisionCmdParser(Command:=PersistentVars.Programs[SelectedProgramNumber].Commands[SelectedRecipeRowIndex].CommandString);
			stVisionCmd := VisionCmdParser.stCommand;
			
		DUT_CommandType.VarSetCommand:
			VarSetCmdParser(Command:=PersistentVars.Programs[SelectedProgramNumber].Commands[SelectedRecipeRowIndex].CommandString);
			stVarSetCmd := VarSetCmdParser.stCommand;
			
		DUT_CommandType.CncCommand:
			CncCmdParser(Command:=PersistentVars.Programs[SelectedProgramNumber].Commands[SelectedRecipeRowIndex].CommandString);
			stCncCmd := CncCmdParser.stCommand;
			
		DUT_CommandType.LogicCommand:
			LogicCmdParser(Command:=PersistentVars.Programs[SelectedProgramNumber].Commands[SelectedRecipeRowIndex].CommandString);
			stLogicCmd := LogicCmdParser.stCommand;
			
	END_CASE
	
END_IF

// should be called after CopySelectedCommand case statement
CurrentVisu := VisuElems.CurrentVisu;
OpenDialog(
	xExecute:= , 
	xDone=> , 
	xBusy=> , 
	xError=> , 
	itfClientFilter:= , 
	eError=> , 
	sDialogName:= , 
	xModal:= TRUE, // TRUE - visu in background cannot be used
	pTopLeftPosition:= , 
	itfDialogOpenedListener:= , 
	pbyDialogInterfaceData:= , 
	udiDialogInterfaceDataSize:= , 
	itfDialogCloseListener:= , 
	pbyTagForDialogClosed:= , 
	dwDialogFlags:= );
IF (OpenDialog.xExecute AND OpenDialog.xDone) 
	OR OpenDialog.xError 
	THEN
		OpenDialog.xExecute := FALSE;
END_IF

// alarms
IF GVL.xClearHistory THEN
    FOR iAlarmCfg := 0 TO AlarmManager.AlarmGlobals.g_AlarmHandler.AlarmConfigurationCount - 1 DO
        itfAlarmConfiguration := AlarmManager.AlarmGlobals.g_AlarmHandler.GetAlarmConfiguration(iAlarmCfg);
        IF __QUERYINTERFACE(itfAlarmConfiguration, itfAlarmConfiguration7) THEN
            itfAlarmConfiguration7.ClearHistory(xKeepActiveAlarms := TRUE); // xKeepActiveAlarms := TRUE so a live fault isn’t ripped out of the recorder.
        END_IF
    END_FOR
    GVL.xClearHistory := FALSE;
END_IF
                  
END_PROGRAM

FUNCTION F_BuildOutputCmd : STRING(GVL.COMMAND_LEN)
VAR_INPUT
	stCommand: ST_OutputCmd;
END_VAR
VAR
    _Command: STRING(GVL.COMMAND_LEN);
END_VAR
VAR CONSTANT
	_Delimiter: STRING:=' ';
	_OutTypeDig: STRING(3):='DIG';
	_OutTypePwm: STRING(3):='PWM';
END_VAR

                    // DIG +0001.00 +0001.00 (turn digital input 1 on)
// DIG +0001.00 +0000.00 (turn digital input 1 off)
// PWM +0001.00 +0030.00(set PWM 1 to position 30)

// clear the command
_Command:='';

//
CASE stCommand.OutputType OF
	DUT_OutputType.Digital:
		F_AddElement(_Command, _Delimiter, _OutTypeDig);
	DUT_OutputType.Pwm:
		F_AddElement(_Command, _Delimiter, _OutTypePwm);
END_CASE

//
F_AddElement(_Command, _Delimiter, INT_TO_STRING(stCommand.OutputTarget));

//
F_AddElement(_Command, _Delimiter, LREAL_TO_STRING(stCommand.OutputValue1));

// set function equal to command
F_BuildOutputCmd := _Command;
                  
END_FUNCTION

FUNCTION_BLOCK FB_ParseOutputCmd
VAR_INPUT
	Command: STRING(GVL.COMMAND_LEN);
END_VAR
VAR_OUTPUT
	stCommand: ST_OutputCmd;
	Error: BOOL;
	ErrorDescription: STRING;
END_VAR
VAR
	_CmdParams: ARRAY [0..GVL.COMMAND_LEN] OF STRING;
	_OutputType: STRING;
END_VAR

                    // DIG +0001.00 +0001.00 (turn digital input 1 on)
// DIG +0001.00 +0000.00 (turn digital input 1 off)
// PWM +0001.00 +0030.00(set PWM 1 to position 30)

Error:=FALSE;
ErrorDescription:='';

// split command string into commands
_CmdParams:=F_SplitCmd(Command:=Command);

_OutputType := _CmdParams[0];
IF _OutputType = 'DIG' THEN
	stCommand.OutputType := DUT_OutputType.Digital;
ELSIF _OutputType = 'PWM' THEN
	stCommand.OutputType := DUT_OutputType.Pwm;
END_IF
stCommand.OutputTarget := STRING_TO_INT(_CmdParams[1]);
stCommand.OutputValue1 := STRING_TO_LREAL(_CmdParams[2]);
                  
END_FUNCTION_BLOCK

FUNCTION F_BuildPauseCmd : STRING(GVL.COMMAND_LEN)
VAR_INPUT
	stCommand: ST_PauseCmd;
END_VAR
VAR
    _Command: STRING(GVL.COMMAND_LEN);
END_VAR
VAR CONSTANT
	_Delimiter: STRING:=' ';
END_VAR

                    // clear the command
_Command:='';

// build command
F_AddElement(_Command, _Delimiter, TIME_TO_STRING(stCommand.PauseTime));

// set function equal to command
F_BuildPauseCmd := _Command;
                  
END_FUNCTION

FUNCTION_BLOCK FB_ParsePauseCmd
VAR_INPUT
	Command: STRING(GVL.COMMAND_LEN);
END_VAR
VAR_OUTPUT
	stCommand: ST_PauseCmd;
	Error: BOOL;
	ErrorDescription: STRING;
END_VAR
VAR
	_CmdParams: ARRAY [0..GVL.COMMAND_LEN] OF STRING;
END_VAR

                    // T#30s

Error:=FALSE;
ErrorDescription:='';

// split command string into commands
_CmdParams:=F_SplitCmd(Command:=Command);

stCommand.PauseTime := STRING_TO_TIME(_CmdParams[0]);
                  
END_FUNCTION_BLOCK

PROGRAM _40_Vision
// vision is separated into its own program so that we can
// assign it to its own core! how awesome is that?!
VAR
	ProcessVisionCommand: FB_VisionCmdProcessor;
   	HostName   : STRING;
	VisionSystemUrl: STRING;
	VisionOutputImageUrl: STRING;
	VisionSystemIpAddress_Last: STRING(19);
    VisionOutputImageScaling: REAL := 1000.0;
    VisionImageWidth: INT:=365; // TODO figure out a way to dynamically set this based on the values set in the visu element properties
    VisionImageHeight: INT:=255;
END_VAR
VAR CONSTANT
	LocalIpAddress: STRING(19):='127.0.0.1';
END_VAR

                    
// used to show the output image on the HMI
// local vision:  http://<plc-hostname>.local:5000/output_sized?width=365&height=255
// remote vision: http://<vision-ip>:5000/output_sized?width=365&height=255
IF PersistentVars.VisionSystemIpAddress <> VisionSystemIpAddress_Last THEN
    VisionSystemIpAddress_Last := PersistentVars.VisionSystemIpAddress;
    //
    IF PersistentVars.VisionSystemIpAddress = LocalIpAddress THEN
        // WebVisu runs in the PC browser, so 127.0.0.1 would hit the PC.
        // Use this PLC's mDNS name instead.
        // https://forge.codesys.com/forge/talk/Runtime/thread/61d60a9fb7/
        SysSockGetHostName(szHostName:=HostName, diNameLen:=SIZEOF(HostName));
        VisionSystemUrl := CONCAT('http://', HostName);
        VisionSystemUrl := CONCAT(VisionSystemUrl, '.local');
    ELSE
        // Dedicated vision Pi: the Programming HMI IP is already that box.
        VisionSystemUrl := CONCAT('http://', PersistentVars.VisionSystemIpAddress);
    END_IF
    //
    VisionSystemUrl := CONCAT(VisionSystemUrl, ':5000/vision');
    VisionOutputImageUrl := CONCAT(VisionSystemUrl,'/output_sized?width=');
    VisionOutputImageUrl := CONCAT(VisionOutputImageUrl,INT_TO_STRING(VisionImageWidth));
    VisionOutputImageUrl := CONCAT(VisionOutputImageUrl,'&height=');
    VisionOutputImageUrl := CONCAT(VisionOutputImageUrl,INT_TO_STRING(VisionImageHeight));
END_IF

//
ProcessVisionCommand(
    VisionSystemIpAddress:= PersistentVars.VisionSystemIpAddress,
    VisionSystemPort:= PersistentVars.VisionSystemPort,
    StoredPositions:= PersistentVars.StoredPositions,
    VisionRegisters:= PersistentVars.VisionRegisters,
    Flags:= PersistentVars.Flags,
    LogicCmdIO:= GVL.CmdIO,
    ItfUnitMode=> ,
    Error=> ,
    ErrorDescription=> ,
    VisionStateText=> );
                  
END_PROGRAM

FUNCTION_BLOCK FB_CncPathPlanner
VAR_IN_OUT
	VarList: SMC_VarList;
END_VAR
VAR_INPUT
END_VAR
VAR_OUTPUT
	DataOut: POINTER TO SMC_OUTQUEUE;
	Busy: BOOL;
	Done: BOOL;
	Error: BOOL;
	ErrorDescription: STRING;
    GcodeText: SMC_GCODE_TEXT;
END_VAR
VAR
	_Filename: STRING := '_cnc/CNC_FromFile.cnc';
	_SMC_ReadNCFile2: SMC_ReadNCFile2;
	_SMC_NCInterpreter: SMC_NCInterpreter;
    _SMC_SmoothPath: SMC_SmoothPath;
	_SMC_CheckVelocities: SMC_CheckVelocities;
	_SMC_GEOINFO_Ipo: ARRAY[0..50] OF SMC_GEOINFO;
	_SMC_GEOINFO_Smooth: ARRAY[0..50] OF SMC_GEOINFO;
	_StartPos: SMC_PosInfo;
	_OriConvention: SMC_ORI_CONVENTION := SMC_ORI_CONVENTION.ZYZ;
	_ExecuteRtrig: R_TRIG;
	_Execute: BOOL;
	_ResetRtrig: R_TRIG;
	_Reset: BOOL;
	_Sequence: INT:=0;
	_ErrorRtrig: R_TRIG;
END_VAR
VAR CONSTANT
	_BaseCncDirectory: STRING:='_cnc/'; // before update to 3.5.19.40 '/var/opt/codesys/_cnc/'
END_VAR

                    _ExecuteRtrig(CLK:=_Execute);
IF _ExecuteRtrig.Q THEN
	_Execute:= FALSE;
END_IF
_ResetRtrig(CLK:=_Reset);
IF _ResetRtrig.Q THEN
	_Reset:= FALSE;
	_Sequence:=999;
END_IF

Busy := _Sequence <> 000;

CASE _Sequence OF
	999:
		_SMC_ReadNCFile2.bExecute := FALSE;
		_Sequence := 000;
	000:
		IF _ExecuteRtrig.Q THEN
			_SMC_ReadNCFile2.bExecute := TRUE;
			_Sequence := 1;
		END_IF
	001:
		IF NOT _SMC_CheckVelocities.bBusy THEN
			_Sequence := 999;
			Done := TRUE;
		END_IF
	
END_CASE

_SMC_ReadNCFile2(
	bExecute:= , 
	bAbort:= _Sequence = 999, 
	sFileName:= _Filename, 
	pvl:= ADR(VarList), 
	fDefaultVel:= , 
	fDefaultAccel:= , 
	fDefaultDecel:= , 
	fDefaultVelFF:= , 
	fDefaultAccelFF:= , 
	fDefaultDecelFF:= , 
	b3DMode:= , 
	bStepSuppress:= , 
	aSubProgramDirs:= , 
	bParenthesesAsComments:= , 
	bDisableJumpBuffer:= , 
	pCustomFunTable:= , 
	aTokenModifier:= , 
	aSentenceModifier:= , 
	bBusy=> , 
	bError=> , 
	ErrorID=> , 
	errorPos=> , 
	ErrorProgramName=> , 
	sentences=> , 
	adwFileSize=> , 
	adwPos=> );

// https://content.helpme-codesys.com/en/libs/SM3_CNC/Current/SM_CNC_POUs/NC2/Interpreter/SMC_NCInterpreter.html
_SMC_NCInterpreter(
	sentences:= _SMC_ReadNCFile2.sentences, 
	bExecute:= _SMC_ReadNCFile2.bExecute, 
	bAbort:= _Sequence = 999, 
	bAppend:= , 
	piStartPosition:= _StartPos, 
	vStartToolLength:= , 
	nSizeOutQueue:= SIZEOF(_SMC_GEOINFO_Ipo), 
	pbyBufferOutQueue:= ADR(_SMC_GEOINFO_Ipo), 
	bEnableSyntaxChecks:= , 
	eOriConv:= _OriConvention,    
    // A/B/C as independent axes so G91 A-45 is signed and can pass ±180.
    // Tracker/trafo stay ZYX; do not set _OriConvention to ADDAXES (that feeds J4/J5/J6 as Euler and faults the group).
    //eOriConv:= SMC_ORI_CONVENTION.ADDAXES,
	dCircleTolerance:= , 
	pInterpreterStack:= , 
	nInterpreterStackSizeBytes:= , 
	bDone=> , 
	bBusy=> , 
	bError=> , 
	wErrorID=> , 
	errorPos=> , 
	poqDataOut=> , 
	iStatus=> , 
	iLineNumberDecoded=> , 
	GCodeText=> GcodeText, 
	CallstackInfo=> , 
	aActivePrograms=> );
    
_SMC_SmoothPath(
	bExecute:= _SMC_ReadNCFile2.bExecute, 
	bAbort:= _Sequence = 999, 
	bAppend:= , 
	poqDataIn:= _SMC_NCInterpreter.poqDataOut, 
	dEdgeDistance:= , 
	dAngleTol:= , 
	nSizeOutQueue:= SIZEOF(_SMC_GEOINFO_Smooth), 
	pbyBufferOutQueue:= ADR(_SMC_GEOINFO_Smooth), 
	eMode:= , 
	bSymmetricalDistances:= , 
	bImprovedSymmetricCuts:= , 
	eAddAxMode:= , 
	dMinimumCurvatureRadius:= , 
	bCheckCurvature:= , 
	dRelativeCurvatureTol:= , 
	bCheckAddAxVelJump:= , 
	dMaxAddAxVelDifference:= , 
	bDone=> , 
	bBusy=> , 
	bError=> , 
	wErrorID=> , 
	poqDataOut=> , 
	udiStopsDueToCurvatureRadius=> );

_SMC_CheckVelocities(
	bExecute:= _SMC_NCInterpreter.bExecute, 
	bAbort:= _Sequence = 999, 
	poqDataIn:= _SMC_SmoothPath.poqDataOut, 
	dAngleTol:= , 
	bCheckAddAxVelJump:= , 
	dMaxAddAxVelDifference:= , 
	bBusy=> , 
	bError=> , 
	wErrorID=> , 
	poqDataOut=> DataOut);
	
_ErrorRtrig();
_ErrorRtrig.CLK:= _SMC_ReadNCFile2.bError
				OR _SMC_NCInterpreter.bError
				OR _SMC_SmoothPath.bError
				OR _SMC_CheckVelocities.bError;
IF _ErrorRtrig.Q THEN
	Error := TRUE;
	IF _SMC_ReadNCFile2.bError THEN
		ErrorDescription := CONCAT(' ReadNCFile Error: ',
                                CONCAT(TO_STRING(_SMC_ReadNCFile2.ErrorID),
                                CONCAT(' ', SMC_ErrorString(_SMC_ReadNCFile2.ErrorID,
                                            SMC_Language_Type.english)))) ;
	END_IF
	IF _SMC_NCInterpreter.bError THEN
		ErrorDescription := CONCAT(' NCInterpreter Error: ',
                                CONCAT(TO_STRING(_SMC_NCInterpreter.wErrorID),
                                CONCAT(' ', SMC_ErrorString(_SMC_NCInterpreter.wErrorID,
                                            SMC_Language_Type.english)))) ;
	END_IF
	IF _SMC_SmoothPath.bError THEN
		ErrorDescription := CONCAT(' SmoothPath Error: ',
                                CONCAT(TO_STRING(_SMC_SmoothPath.wErrorID),
                                CONCAT(' ', SMC_ErrorString(_SMC_SmoothPath.wErrorID,
                                            SMC_Language_Type.english)))) ;
	END_IF
	IF _SMC_CheckVelocities.bError THEN
		ErrorDescription := CONCAT(' CheckVelocities Error: ',
                                CONCAT(TO_STRING(_SMC_CheckVelocities.wErrorID),
                                CONCAT(' ', SMC_ErrorString(_SMC_CheckVelocities.wErrorID,
                                            SMC_Language_Type.english)))) ;
	END_IF
END_IF
                  

METHOD PUBLIC M_Execute : BOOL
VAR_INPUT
	Filename: STRING := 'CNC_FromFile.cnc';
END_VAR
                          _Filename := CONCAT(_BaseCncDirectory, Filename);
_Execute:=TRUE;
Done := FALSE;
                        
END_METHOD

METHOD PUBLIC M_Reset : BOOL
VAR_INPUT
END_VAR
                          _Reset := TRUE;
Error := FALSE;
ErrorDescription := '';
                        
END_METHOD

METHOD PUBLIC M_SetStartPosition : BOOL
VAR_INPUT
	StartPos: SMC_PosInfo;
END_VAR
                          _StartPos := StartPos;
                        
END_METHOD

METHOD PUBLIC M_SetOriConvention : BOOL
VAR_INPUT
	OriConvention: SMC_ORI_CONVENTION := SMC_ORI_CONVENTION.ZYZ;
END_VAR
                          _OriConvention := OriConvention;
GVL.OriConvention := OriConvention;
                        
END_METHOD
END_FUNCTION_BLOCK

FUNCTION F_BuildCncCmd : STRING(GVL.COMMAND_LEN)
VAR_INPUT
	stCommand: ST_CncCmd;
END_VAR
VAR
	_Command: STRING(GVL.COMMAND_LEN);
END_VAR
VAR CONSTANT
	_Delimiter: STRING:=' ';
	_AddString: STRING(3):='ADD';
	_XYZString: STRING(3):='XYZ';
	_ZYXString: STRING(3):='ZYX';
	_ZYZString: STRING(3):='ZYZ';
	_LiteralString: STRING(3):='LIT';
	_VariableString: STRING(3):='VAR';
	_StoredPositionsString: STRING(3):='STO';
	_VisionRegistersString: STRING(3):='VIS';
	_FlagsString: STRING(3):='FLG';
END_VAR

                    // /path/to/file/with/no/spaces/file.cnc ADD|XYX|ZYX|ZYZ startpos
// file1.cnc XYZ H +0250.00 +0000.00 +0500.00 +0000.00 +0045.00 +0180.00
// file2.cnc ADD A S 025
// file3.cnc ADD A V 015

// note: the command format will only contain the filename moving forward until the issues with the transformation function blocks gets resolved by CODESYS. See notes in the CncCommandProcessor about this.
// file3.cnc 

_Command:='';

//
F_AddElement(_Command, _Delimiter, stCommand.Filename);

//
(*CASE stCommand.OriConvention OF
	SMC_ORI_CONVENTION.ADDAXES:
		F_AddElement(_Command, _Delimiter, _AddString);
	SMC_ORI_CONVENTION.XYZ:
		F_AddElement(_Command, _Delimiter, _XYZString);
	SMC_ORI_CONVENTION.ZYX:
		F_AddElement(_Command, _Delimiter, _ZYXString);
	SMC_ORI_CONVENTION.ZYZ:
		F_AddElement(_Command, _Delimiter, _ZYZString);
END_CASE

//
CASE stCommand.CoordinateType OF
	DUT_Command_CoordinateType.Literal:
		F_AddElement(_Command, _Delimiter, _LiteralString);
		F_AddElement(_Command, _Delimiter, LREAL_TO_STRING(stCommand.StartPos.dX));
		F_AddElement(_Command, _Delimiter, LREAL_TO_STRING(stCommand.StartPos.dY));
		F_AddElement(_Command, _Delimiter, LREAL_TO_STRING(stCommand.StartPos.dZ));
		F_AddElement(_Command, _Delimiter, LREAL_TO_STRING(stCommand.StartPos.dA));
		F_AddElement(_Command, _Delimiter, LREAL_TO_STRING(stCommand.StartPos.dB));
		F_AddElement(_Command, _Delimiter, LREAL_TO_STRING(stCommand.StartPos.dC));
		
	DUT_Command_CoordinateType.Variable:
		F_AddElement(_Command, _Delimiter, _VariableString);
		CASE stCommand.ArrayType OF
			DUT_Command_ArrayType.StoredPosition:
				F_AddElement(_Command, _Delimiter, _StoredPositionsString);
			DUT_Command_ArrayType.VisionRegister:
				F_AddElement(_Command, _Delimiter, _VisionRegistersString);
			DUT_Command_ArrayType.Flag:
				F_AddElement(_Command, _Delimiter, _FlagsString);
		END_CASE
		F_AddElement(_Command, _Delimiter, INT_TO_STRING(stCommand.ArrayIndex));
		
END_CASE*)

F_BuildCncCmd := _Command;

                  
END_FUNCTION

FUNCTION_BLOCK FB_PositionTracker
VAR_IN_OUT
	AxisGroup: AXIS_GROUP_REF_SM3;
	J1: AXIS_REF_SM3;
	J2: AXIS_REF_SM3;
	J3: AXIS_REF_SM3;
	J4: AXIS_REF_SM3;
	J5: AXIS_REF_SM3;
	J6: AXIS_REF_SM3;
END_VAR
VAR_INPUT
    OriConvention: SMC_ORI_CONVENTION := SMC_ORI_CONVENTION.ZYZ;
END_VAR
VAR_OUTPUT
	VisuStruct3DTrack: VisuStruct3DTrack;
    Position: SMC_PosInfo;
	Arm: SMC_ArticulatedRobot_6DOF_J0_State;
	Elbow: SMC_ArticulatedRobot_6DOF_J1_State;
	Hand: SMC_ArticulatedRobot_6DOF_J4_State;
END_VAR
VAR
	_SMC_TrafoConfig_ArticulatedRobot_6DOF: SMC_TrafoConfig_ArticulatedRobot_6DOF;
	_SMC_Trafo_ArticulatedRobot_6DOF: SMC_Trafo_ArticulatedRobot_6DOF;
	_SMC_Trafof_ArticulatedRobot_6DOF: SMC_Trafof_ArticulatedRobot_6DOF;
	_VisuStruct3DPathPoint: ARRAY [0..5000] OF VisuStruct3DPathPoint;
	_SMC_PositionTracker: SMC_PositionTracker;
	_PositionTrackerClearR_Trig: R_Trig;
	_Clear: BOOL:=FALSE;
END_VAR

                    
// NOTE currently the settings for J6 invert direction under scaling/mapping contradict using motion control 
// libraries and CNC. For CNC to work properly, the setting is required to be enabled (inverted). Additionally
// the homing direction and position will need to be negated. This all requires a full download. Will be leaving 
// setting disabled for now so that we can continue to use motion control. 
//
// to recap, take these steps if you would like to try out CNC:
// 1. open the axis pool settings and under the scaling/mapping section enable 'invert direction'
// 2. in the A_Homing POU, change the homing direction to positive.
// 3. in _00_MAIN POU, under FirstScan set the initial home offset to a positive value (keep the value and just change the sign).
// 4. do a full download.
// 5. go online and set the persistent value (if previously initialized in FirstScan) to a positive value.
//
// UPDATE: Figured out a work around for this issue. In the A_Interpolater POU, I negated the set position in the ControlAxisByPos
// function block for J6 such that it drives the opposite way. This appears to have resolved the issue. Why this is needed, I do not
// know. I am sure it is some minor overlooked detail somewhere in the code...


_SMC_TrafoConfig_ArticulatedRobot_6DOF.a1:=ArfBotAxisGroup.Trafo.a1;//AxisGroup.Trafo.a1;
_SMC_TrafoConfig_ArticulatedRobot_6DOF.a2:=ArfBotAxisGroup.Trafo.a2;//AxisGroup.Trafo.a2;
_SMC_TrafoConfig_ArticulatedRobot_6DOF.a3:=ArfBotAxisGroup.Trafo.a3;//AxisGroup.Trafo.a3;
// conflicting documentation on if d1 needs to be pos or neg. only works as negative otherwise trafo reports invalid configuration
// https://product-help.schneider-electric.com/Machine%20Expert/V2.0/zh/codesys_softmotion/codesys_softmotion/modules/_sm_trafo_pou_six_dof_robot.html
// https://forge.codesys.com/forge/talk/Motion/thread/16e1f0327f/
_SMC_TrafoConfig_ArticulatedRobot_6DOF.d1:=-ArfBotAxisGroup.Trafo.d1;//-AxisGroup.Trafo.d1;
_SMC_TrafoConfig_ArticulatedRobot_6DOF.d3:=ArfBotAxisGroup.Trafo.d3;//AxisGroup.Trafo.d3;
_SMC_TrafoConfig_ArticulatedRobot_6DOF.d4:=ArfBotAxisGroup.Trafo.d4;//AxisGroup.Trafo.d4;
_SMC_TrafoConfig_ArticulatedRobot_6DOF.d6:=ArfBotAxisGroup.Trafo.d6;//AxisGroup.Trafo.d6;
_SMC_TrafoConfig_ArticulatedRobot_6DOF.q3_max_deg:=160; // TODO put magic numbers somewhere appropriate
_SMC_TrafoConfig_ArticulatedRobot_6DOF.q3_min_deg:=-160; // TODO put magic numbers somewhere appropriate
_SMC_TrafoConfig_ArticulatedRobot_6DOF.q5_max_deg:=160; // TODO put magic numbers somewhere appropriate
_SMC_TrafoConfig_ArticulatedRobot_6DOF.q5_min_deg:=-160; // TODO put magic numbers somewhere appropriate

// track position
_SMC_Trafof_ArticulatedRobot_6DOF(config:=_SMC_TrafoConfig_ArticulatedRobot_6DOF,
							Drive0:=J1,
							Drive1:=J2,
							Drive2:=J3,
							Drive3:=J4,
							Drive4:=J5,
							Drive5:=J6,
							vToolPos=>,
							mToolOrientation=>,
							armState=>Arm,
							elbowState=>Elbow,
							handState=>Hand);
Position.dX := _SMC_Trafof_ArticulatedRobot_6DOF.vToolPos.dX;
Position.dY := _SMC_Trafof_ArticulatedRobot_6DOF.vToolPos.dY;
Position.dZ := _SMC_Trafof_ArticulatedRobot_6DOF.vToolPos.dZ;

// https://content.helpme-codesys.com/en/libs/SM3_Math/4.12.0.0/Matrix3/fld-Matrix3.html
// ATTENTION: ZYZ is the only orientation convention that was reliable during testing.
CASE OriConvention OF
    SMC_ORI_CONVENTION.ADDAXES:
        Position.dA := J4.fActPosition;
        Position.dB := J5.fActPosition;
        Position.dC := J6.fActPosition;
    SMC_ORI_CONVENTION.XYZ:
        SMC_Matrix3_ToRollPitchYaw_deg( mR:=_SMC_Trafof_ArticulatedRobot_6DOF.mToolOrientation, 
                                        dRoll=> Position.dA, dPitch=> Position.dB, dYaw=> Position.dC);
    SMC_ORI_CONVENTION.ZYX:
        // yaw(Z), pitch(Y) and roll(X)
        SMC_Matrix3_ToYawPitchRoll( mR:=_SMC_Trafof_ArticulatedRobot_6DOF.mToolOrientation, 
                                    dYaw_rad=> Position.dA, dPitch_rad=> Position.dB, dRoll_rad=> Position.dC);
                                    Position.dA := F_RadToDeg(Position.dA);
                                    Position.dB := F_RadToDeg(Position.dB);
                                    Position.dC := F_RadToDeg(Position.dC);
    SMC_ORI_CONVENTION.ZYZ:
        SMC_Matrix3_ToZYZ_deg(  mR:=_SMC_Trafof_ArticulatedRobot_6DOF.mToolOrientation, 
                                dA_deg=> Position.dA, dB_deg=> Position.dB, dC_deg=> Position.dC);
END_CASE

_PositionTrackerClearR_Trig(Clk:=_Clear);
_SMC_PositionTracker(
	bEnable:= TRUE, 
	bClear:= _PositionTrackerClearR_Trig.Q, 
	dX:= _SMC_Trafof_ArticulatedRobot_6DOF.vToolPos.dX, 
	dY:= _SMC_Trafof_ArticulatedRobot_6DOF.vToolPos.dY, 
	dZ:= _SMC_Trafof_ArticulatedRobot_6DOF.vToolPos.dZ, 
	udiNumberOfPointsInArray:= SIZEOF(_VisuStruct3DPathPoint) / SIZEOF(VisuStruct3DPathPoint), 
	pBuffer:= ADR(_VisuStruct3DPathPoint), 
	vs3dt=> VisuStruct3DTrack);
_Clear := FALSE;
                  

METHOD PUBLIC M_Clear
VAR_INPUT
END_VAR
                          _Clear := TRUE;
                        
END_METHOD
END_FUNCTION_BLOCK

FUNCTION_BLOCK FB_OpenCV EXTENDS FB_PythonServerHandler
VAR_INPUT
END_VAR
VAR_OUTPUT
END_VAR
VAR
END_VAR

                    SUPER^();
                  

METHOD PUBLIC M_CalibrateCamera : BOOL
VAR_INPUT
	iImageWidth: UINT:=2016;
	iImageHeight: UINT:=2000;
	uTimeout: UDINT:=60; //sec
	fCalCheckerSize: REAL:=25.0; //mm
	iCalCheckerX: UINT:=6;
	iCalCheckerY: UINT:=9;
END_VAR
VAR
	_Command : STRING(255);
END_VAR
VAR	
	_CalScriptFileName: STRING:='/var/opt/codesys/PlcLogic/Application/Vision/CalibrateCamera.py';
	_CalResultFile: STRING:='/var/opt/codesys/PlcLogic/visu/outputimage.jpg';
END_VAR
                          
// calibrate with a checkerboard
// sudo python /var/opt/codesys/PlcLogic/Application/CalibrateCamera.py -s cal.yaml -l 24.5 -x 6 -y 9 -d false

IF NOT _Busy THEN
	M_CalibrateCamera := TRUE;
	
	_Command := CONCAT('sudo python ', _CalScriptFileName);
	_Command := CONCAT(_Command, ' -l ');
	_Command := CONCAT(_Command, REAL_TO_STRING(fCalCheckerSize));
	_Command := CONCAT(_Command, ' -x ');
	_Command := CONCAT(_Command, UINT_TO_STRING(iCalCheckerX));
	_Command := CONCAT(_Command, ' -y ');
	_Command := CONCAT(_Command, UINT_TO_STRING(iCalCheckerY));
	_Command := CONCAT(_Command, ' -w ');
	_Command := CONCAT(_Command, UINT_TO_STRING(iImageWidth));
	_Command := CONCAT(_Command, ' -h ');
	_Command := CONCAT(_Command, UINT_TO_STRING(iImageHeight));
	_Command := CONCAT(_Command, ' -r ');
	_Command := CONCAT(_Command, _CalResultFile);
	_Command := CONCAT(_Command, ' 2> ./vision_log.txt ');
	
	SUPER^._M_Execute(Command:=_Command, Timeout:=uTimeout);
	
ELSE
	M_CalibrateCamera := FALSE;
	//_Error := TRUE;
	//_ErrorDescription := 'function busy.';
	
END_IF
                        
END_METHOD

METHOD PUBLIC M_CaptureImage : BOOL
VAR_INPUT
	iImageWidth: UINT:=2016;
	iImageHeight: UINT:=2000;
	uTimeout: UDINT:=60; //sec
END_VAR
VAR
	_Command : STRING(255);
END_VAR
VAR
	_ImageScriptFileName: STRING:='/var/opt/codesys/PlcLogic/Application/Vision/CaptureImage.py';
	_CaptureImageName: STRING:='/var/opt/codesys/PlcLogic/visu/outputimage.jpg';
END_VAR
                          
// capture an image
// sudo python /var/opt/codesys/PlcLogic/Application/CaptureImage.py -s /var/opt/codesys/PlcLogic/Application/input.jpg -w 2016 -h 2000

IF NOT _Busy THEN
	M_CaptureImage := TRUE;
	
	_Command := CONCAT('sudo python ', _ImageScriptFileName);
	_Command := CONCAT(_Command, ' -s ');
	_Command := CONCAT(_Command, _CaptureImageName);
	_Command := CONCAT(_Command, ' -w ');
	_Command := CONCAT(_Command, UINT_TO_STRING(iImageWidth));
	_Command := CONCAT(_Command, ' -h ');
	_Command := CONCAT(_Command, UINT_TO_STRING(iImageHeight));
	_Command := CONCAT(_Command, ' 2> ./vision_log.txt ');
	
	SUPER^._M_Execute(Command:=_Command, Timeout:=uTimeout);
	
ELSE
	M_CaptureImage := FALSE;
	//_Error := TRUE;
	//_ErrorDescription := 'function busy.';
	
END_IF

                        
END_METHOD

METHOD PUBLIC M_LocatePart : BOOL
VAR_INPUT
	iImageWidth: UINT:=2016;
	iImageHeight: UINT:=2000;
	uTimeout: UDINT:=60; //sec
	iMaxPos: UINT:=10; // i
	dMaxOverlap: REAL:=0.0; // j
	dScore: REAL:=0.8; // k
	dToleranceAngle: REAL:=90.0; // l
	sTemplateName: STRING:='template.jpg';
	sScriptFilename: STRING:='FastTemplateMatching.py';
END_VAR
VAR
	_Command : STRING(255);
END_VAR
VAR CONSTANT
	//_SCRIPT_FILE_NAME: STRING:='/var/opt/codesys/PlcLogic/Application/Vision/FastTemplateMatching.py';
	_SCRIPT_DIR_PATH: STRING:='/var/opt/codesys/PlcLogic/Application/Vision/';
	_RESULT_FILE_NAME: STRING:='/var/opt/codesys/PlcLogic/visu/outputimage.jpg';
	_TEMPLATE_DIR_PATH: STRING:='/var/opt/codesys/PlcLogic/Application/Vision/Templates/';
END_VAR
                          
// run the designated vision program
// sudo python /var/opt/codesys/PlcLogic/Application/Vision/TemplateMatch.py -s /var/opt/codesys/PlcLogic/visu/outputimage.jpg        -t /var/opt/codesys/PlcLogic/Application/Vision/Template3.JPG -i 0.9 -j 1.0 -d true -w 2016 -h 2000
// sudo python /var/opt/codesys/PlcLogic/Application/Vision/FastTemplateMatching.py -s /var/opt/codesys/PlcLogic/visu/outputimage.jpg -t /var/opt/codesys/PlcLogic/Application/Vision/Template.jpg -w 2016 -h 2000 -d false
IF NOT _Busy THEN
	M_LocatePart := TRUE;
	
	_Command := CONCAT('sudo python ', _SCRIPT_DIR_PATH);
	_Command := CONCAT(_Command, sScriptFilename);
	//_Command := CONCAT(_Command, ' -s '); // need to trim down the string length
	//_Command := CONCAT(_Command, _VisionImageName);
	_Command := CONCAT(_Command, ' -t ');
	_Command := CONCAT(_Command, _TEMPLATE_DIR_PATH);
	_Command := CONCAT(_Command, sTemplateName);
	_Command := CONCAT(_Command, ' -i ');
	_Command := CONCAT(_Command, UINT_TO_STRING(iMaxPos));
	_Command := CONCAT(_Command, ' -j ');
	_Command := CONCAT(_Command, REAL_TO_STRING(dMaxOverlap));
	_Command := CONCAT(_Command, ' -k ');
	_Command := CONCAT(_Command, REAL_TO_STRING(dScore));
	_Command := CONCAT(_Command, ' -l ');
	_Command := CONCAT(_Command, REAL_TO_STRING(dToleranceAngle));
	_Command := CONCAT(_Command, ' -w ');
	_Command := CONCAT(_Command, UINT_TO_STRING(iImageWidth));
	_Command := CONCAT(_Command, ' -h ');
	_Command := CONCAT(_Command, UINT_TO_STRING(iImageHeight));
	_Command := CONCAT(_Command, ' 2> ./vision_log.txt ');
	
	SUPER^._M_Execute(Command:=_Command, Timeout:=uTimeout);
	
ELSE
	M_LocatePart := FALSE;
	//_Error := TRUE;
	//_ErrorDescription := 'function busy.';
	
END_IF
                        
END_METHOD
END_FUNCTION_BLOCK

FUNCTION_BLOCK FB_TcpClient
VAR_INPUT
	bEnable: BOOL;
	strIpAddress: STRING(19):='127.0.0.1';
	uPort: UINT:=50011;
END_VAR
VAR
	_Write: BOOL:=FALSE;
	_DataToWrite: STRING(255):='';
END_VAR
VAR_OUTPUT
	bBusyWrite: BOOL;
	bDoneWrite: BOOL;
	bBusyRead: BOOL;
	dRecordRead: DINT;
	strRead: STRING(255);
	byteArrayRead: ARRAY[0..254] OF BYTE;
	bConnected: BOOL;
END_VAR

VAR
{warning disable C0540}
    _ipAddress       : NBS.IPv4Address;
{warning restore C0540}
    _fbTcpClient     : NBS.TCP_Client;
    _fbTcpRead       : NBS.TCP_Read;
    _fbTcpWrite      : NBS.TCP_Write;	
	
	_ConnectDelayTimer: TON;
	
	_WriteData: StringByteArray;
	_ReadData: StringByteArray;
	
	_WriteRTRIG: R_TRIG;
	_ConnectStep, _ReadStep: INT;
	_Read: BOOL;
END_VAR

VAR CONSTANT
	ConnectStep_IDLE: 	INT:=00;
	ConnectStep_DELAY: 	INT:=10;
	ConnectStep_SETUP: 	INT:=20;
	ConnectStep_ENABLE: INT:=30;
	ConnectStep_WAIT: 	INT:=40;
	ConnectStep_CONN: 	INT:=50;
END_VAR

VAR CONSTANT
	WriteStep_IDLE: 	INT:=00;
	WriteStep_DATA: 	INT:=10;
	WriteStep_WRITE: 	INT:=20;
	WriteStep_WAIT: 	INT:=30;
END_VAR

VAR CONSTANT
	ReadStep_RESET: 	INT:=00;
	ReadStep_IDLE: 		INT:=10;
	ReadStep_ENABLE: 	INT:=20;
	ReadStep_MONITOR: 	INT:=30;
END_VAR

                    {region "connect"}
	
	bConnected := (_ConnectStep = ConnectStep_CONN);
	_ConnectDelayTimer(IN:=_ConnectStep = ConnectStep_DELAY, PT:=T#1S);
	CASE _ConnectStep OF
		
		ConnectStep_IDLE: // IDLE
			IF bEnable THEN
				_fbTcpClient.xEnable := FALSE;
				_ConnectStep := ConnectStep_DELAY;
			END_IF
			
		ConnectStep_DELAY: // DELAY
			IF _ConnectDelayTimer.Q THEN
				_ConnectStep := ConnectStep_SETUP;
			END_IF
			
		ConnectStep_SETUP: // SETUP
			_ipAddress.SetInitialValue(ipAddress := strIpAddress);
			_ConnectStep := ConnectStep_ENABLE;
			
		ConnectStep_ENABLE: // ENABLE
			_fbTcpClient.xEnable := TRUE;
			_ConnectStep := ConnectStep_WAIT;
			
		ConnectStep_WAIT: // WAIT
			IF _fbTcpClient.xActive THEN
				_ConnectStep := ConnectStep_CONN;
			ELSIF _fbTcpClient.xError THEN
				_ConnectStep := ConnectStep_IDLE;
			END_IF
		
		ConnectStep_CONN: // CONNECTED
			IF _fbTcpClient.xError OR NOT _fbTcpClient.xActive OR NOT bEnable THEN
				_ConnectStep := ConnectStep_IDLE;
			END_IF
			
	END_CASE
	
	_fbTcpClient(
		xEnable := , 
		itfIPAddress := _ipAddress, 
		uiPort := uPort, 
		udiTimeOut := 1000000); // us
			 
{endregion}


{region "write"}
	_WriteRTRIG(CLK:=_Write);
	IF _WriteRTRIG.Q THEN
		_Write := FALSE;
		IF bConnected AND _DataToWrite <> '' THEN
			MemUtils.MemSet(	pbyBuffer:=ADR(_WriteData.bArray),
								byValue:=0,
								dwSize:=SIZEOF(_WriteData.bArray));
			MemUtils.MemCpy(	pbyDest:=ADR(_WriteData.sString),
								pbySrc:=ADR(_DataToWrite),
								dwSize:=INT_TO_DWORD(LEN(_DataToWrite)));
			_fbTcpWrite.xExecute := TRUE;
		END_IF
	END_IF
	
	_fbTcpWrite(xExecute := _fbTcpWrite.xExecute AND NOT _fbTcpWrite.xDone AND NOT _fbTcpWrite.xError,
				xBusy=>bBusyWrite,
				xDone=>bDoneWrite,
				itfConnection := _fbTcpClient.itfConnection, 
				udiTimeOut := 1000000, // us 
				udiSize := INT_TO_UDINT(LEN(_WriteData.sString)), 
				pData := ADR(_WriteData.bArray));

{endregion}


{region "read"}

	_Read := (_ConnectStep = ConnectStep_CONN);
	CASE _ReadStep OF
			 
		ReadStep_RESET: // RESET
			_fbTcpRead.xEnable := FALSE;
			_ReadStep := ReadStep_IDLE;

		ReadStep_IDLE: // IDLE
			IF _Read THEN
				_ReadStep := ReadStep_ENABLE;
			END_IF

		ReadStep_ENABLE: // ENABLE
			_fbTcpRead.xEnable := TRUE;
			_ReadStep := ReadStep_MONITOR;

		ReadStep_MONITOR: // MONITOR
			IF _fbTcpRead.xReady THEN
				IF (_fbTcpRead.udiCount > 0) THEN
					//
					MemUtils.MemSet(
						pbyBuffer:=ADR(strRead),
						byValue:=0,
						dwSize:=SIZEOF(strRead)); 
					MemUtils.MemSet(
						pbyBuffer:=ADR(byteArrayRead),
						byValue:=0,
						dwSize:=SIZEOF(byteArrayRead)); 
					MemUtils.MemCpy(
						pbyDest:=ADR(strRead),
						pbySrc:=ADR(_ReadData.sString),
						dwSize:=SEL(_fbTcpRead.udiCount > 255, _fbTcpRead.udiCount, 255));
					MemUtils.MemCpy(
						pbyDest:=ADR(byteArrayRead),
						pbySrc:=ADR(_ReadData.bArray),
						dwSize:=SEL(_fbTcpRead.udiCount > 255, _fbTcpRead.udiCount, 255));
					MemUtils.MemSet(
						pbyBuffer:=ADR(_ReadData.sString),
						byValue:=0,
						dwSize:=SIZEOF(_ReadData.sString)); 
					//
					dRecordRead := dRecordRead + 1;
				END_IF
				
			ELSIF _fbTcpRead.xError OR NOT _Read THEN
				_ReadStep := ReadStep_RESET;
				
			END_IF
			 
	END_CASE
	
	bBusyRead := (_ReadStep <> ReadStep_IDLE) AND _fbTcpRead.xBusy;
	_fbTcpRead(xEnable := , 
				itfConnection := _fbTcpClient.itfConnection, 
				udiSize := SIZEOF(_ReadData.bArray), 
				pData := ADR(_ReadData.bArray), 
				udiCount => );

{endregion}
                  

METHOD INTERNAL _M_Write : BOOL
VAR_INPUT
	Data: STRING(255);
END_VAR
                          IF bConnected AND NOT bBusyWrite THEN
	bBusyWrite := TRUE; // do this as a workaround to show "busy" ASAP to let callers know to hold back
	_Write:=TRUE;
	_DataToWrite:=Data;
	_M_Write := TRUE;
	
ELSE
	_M_Write := FALSE;
	
END_IF
                        
END_METHOD

METHOD INTERNAL _M_Reconnect : BOOL
VAR_INPUT
END_VAR
                          _ConnectStep := ConnectStep_IDLE;
                        
END_METHOD
END_FUNCTION_BLOCK

FUNCTION_BLOCK FB_ParseVisionCmd
VAR_INPUT
    Command: STRING(GVL.COMMAND_LEN);
END_VAR
VAR_OUTPUT
    stCommand: ST_VisionCmd;
	Error: BOOL;
	ErrorDescription: STRING;
END_VAR
VAR
	_CmdParams: ARRAY [0..GVL.COMMAND_LEN] OF STRING;
    _CommandType: STRING;
	_StrPosition: INT;
END_VAR
VAR CONSTANT
	_CommandTypeCal: STRING(3):='CAL'; // calibrate vision
	_CommandTypeCap: STRING(3):='CAP'; // capture image
	_CommandTypeAcq: STRING(3):='ACQ'; // legacy alias for CAP
	_CommandTypeLoc: STRING(3):='LOC'; // locate part
END_VAR

                    // CAL|CAP|LOC ImageWidth ImageHeight Timeout

// CAL Calibrate vision system
    // CheckerSize (user units) XCount YCount 
    // CAL 2016 2000 60 25.0 6 9
    
// CAP Capture image
    // CAP 2016 2000 60
    // ACQ is still accepted as a legacy alias
    
// LOC Locate part 
    // MaxParts MaxOverlap Score ToleranceAngle ResultPostion TemplateName ScriptName
    // LOC 2016 2000 60 10 0.0 0.8 90.0 1 template.jpg FastTemplateMatching.py
	// MaxParts - max number of parts to find in image
	// MaxOverlap - max overlap of parts in image
	// Score - min required score for parts
	// ToleranceAngle - +/- search angle (the larger the number, the longer the search)
	// ResultPostion - index of vision register to store result
	// TemplateName - name of the template to search for
	// ScriptName - name of the template to search for

Error:=FALSE;
ErrorDescription:='';

// split command string into commands
_CmdParams:=F_SplitCmd(Command:=Command);

_CommandType:= _CmdParams[0];
IF _CommandType = _CommandTypeCal THEN
    // CAL 2016 2000 0060 025.0 0006 0009
	stCommand.CommandType:=DUT_Command_VisionType.Calibrate;
    stCommand.Calibrate.CheckerSize:=STRING_TO_REAL(_CmdParams[4]);
    stCommand.Calibrate.CheckerXCount:=STRING_TO_UINT(_CmdParams[5]);
    stCommand.Calibrate.CheckerYCount:=STRING_TO_UINT(_CmdParams[6]);
	
	IF stCommand.Calibrate.CheckerSize <= 0
		OR stCommand.Calibrate.CheckerXCount <= 0
		OR stCommand.Calibrate.CheckerYCount <= 0 THEN
			Error:=TRUE;
			ErrorDescription:='Checkerboard configuration incorrect';
			RETURN;
	END_IF
    
ELSIF (_CommandType = _CommandTypeCap) OR (_CommandType = _CommandTypeAcq) THEN
    // CAP 2016 2000 0060
	stCommand.CommandType:=DUT_Command_VisionType.Capture;
    
ELSIF _CommandType = _CommandTypeLoc THEN
    // LOC 2016 2000 0060 0010 000.0 0.8 090.0 001 template.jpg FastTemplatMatching.py
	stCommand.CommandType:=DUT_Command_VisionType.LocatePart;
    stCommand.Locate.MaxParts:=STRING_TO_UINT(_CmdParams[4]);
    stCommand.Locate.MaxOverlap:=STRING_TO_REAL(_CmdParams[5]);
    stCommand.Locate.Score:=STRING_TO_REAL(_CmdParams[6]);
    stCommand.Locate.ToleranceAngle:=STRING_TO_REAL(_CmdParams[7]);
    stCommand.Locate.ResultPosition:=STRING_TO_UINT(_CmdParams[8]);
    stCommand.Locate.TemplateName:=_CmdParams[9];
    stCommand.Locate.ScriptFilename:=_CmdParams[10];
	
	IF stCommand.Locate.MaxParts <= 0
		OR stCommand.Locate.ResultPosition < GVL.VIS_ARR_BEG
		OR stCommand.Locate.ResultPosition > GVL.VIS_ARR_END
		OR stCommand.Locate.TemplateName = '' THEN
			Error:=TRUE;
			ErrorDescription:='Locate part configuration incorrect';
			RETURN;
	END_IF
	
ELSE
	Error:=TRUE;
	ErrorDescription:='Unknown command type for vision';
	RETURN;
    
END_IF

// common
stCommand.ImageWidth:=STRING_TO_UINT(_CmdParams[1]);
stCommand.ImageHeight:=STRING_TO_UINT(_CmdParams[2]);
stCommand.Timeout:=STRING_TO_UDINT(_CmdParams[3]);

IF stCommand.ImageWidth <= 0
	OR stCommand.ImageHeight <= 0 THEN
		Error:=TRUE;
		ErrorDescription:='Image size settings incorrect';
END_IF
                  
END_FUNCTION_BLOCK

FUNCTION F_BuildVisionCmd : STRING(GVL.COMMAND_LEN)
VAR_INPUT
    stCommand: ST_VisionCmd;
END_VAR
VAR
    _Command: STRING(GVL.COMMAND_LEN);
END_VAR
VAR CONSTANT
	_Delimiter: STRING:=' ';
	_CommandTypeCal: STRING(3):='CAL'; // calibrate vision
	_CommandTypeCap: STRING(3):='CAP'; // capture image
	_CommandTypeLoc: STRING(3):='LOC'; // locate part
END_VAR

                    // CAL|CAP|LOC ImageWidth ImageHeight Timeout

// CAL Calibrate vision system
    // CheckerSize (user units) XCount YCount 
    // CAL 2016 2000 60 25.0 6 9
    
// CAP Capture image
    // CAP 2016 2000 60
    
// LOC Locate part 
    // MaxParts MaxOverlap Score ToleranceAngle ResultPostion TemplateName ScriptName
    // LOC 2016 2000 60 10 0.0 0.8 90.0 1 template.jpg FastTemplateMatching.py
	// MaxParts - max number of parts to find in image
	// MaxOverlap - max overlap of parts in image
	// Score - min required score for parts
	// ToleranceAngle - +/- search angle (the larger the number, the longer the search)
	// ResultPostion - index of vision register to store result
	// TemplateName - name of the template to search for
	// ScriptName - name of the template to search for

// clear the command
_Command:='';

// build the command
CASE stCommand.CommandType OF
	DUT_Command_VisionType.Calibrate:
		F_AddElement(_Command, _Delimiter, _CommandTypeCal);
	DUT_Command_VisionType.Capture:
		F_AddElement(_Command, _Delimiter, _CommandTypeCap);
	DUT_Command_VisionType.LocatePart:
		F_AddElement(_Command, _Delimiter, _CommandTypeLoc);
END_CASE

// add the common items width, height, timeout
F_AddElement(_Command, _Delimiter, UINT_TO_STRING(stCommand.ImageWidth));
F_AddElement(_Command, _Delimiter, UINT_TO_STRING(stCommand.ImageHeight));
F_AddElement(_Command, _Delimiter, UDINT_TO_STRING(stCommand.Timeout));

//
CASE stCommand.CommandType OF
	DUT_Command_VisionType.Calibrate:
		// CAL 2016 2000 60 25.0 6 9
		F_AddElement(_Command, _Delimiter, REAL_TO_STRING(stCommand.Calibrate.CheckerSize));
		F_AddElement(_Command, _Delimiter, UINT_TO_STRING(stCommand.Calibrate.CheckerXCount));
		F_AddElement(_Command, _Delimiter, UINT_TO_STRING(stCommand.Calibrate.CheckerYCount));
		
	DUT_Command_VisionType.Capture:
		// CAP 2016 2000 60
		// we are done
		
	DUT_Command_VisionType.LocatePart:
		// LOC 2016 2000 60 10 0.0 0.8 90.0 1 template.jpg FastTemplateMatching.py
		F_AddElement(_Command, _Delimiter, UINT_TO_STRING(stCommand.Locate.MaxParts));
		F_AddElement(_Command, _Delimiter, REAL_TO_STRING(stCommand.Locate.MaxOverlap));
		F_AddElement(_Command, _Delimiter, REAL_TO_STRING(stCommand.Locate.Score));
		F_AddElement(_Command, _Delimiter, REAL_TO_STRING(stCommand.Locate.ToleranceAngle));
		F_AddElement(_Command, _Delimiter, UINT_TO_STRING(stCommand.Locate.ResultPosition));
		F_AddElement(_Command, _Delimiter, stCommand.Locate.TemplateName);
		F_AddElement(_Command, _Delimiter, stCommand.Locate.ScriptFilename);
		
END_CASE

// set function equal to command
F_BuildVisionCmd := _Command;
                  
END_FUNCTION

FUNCTION_BLOCK FB_Module EXTENDS FB_PackML IMPLEMENTS ItfModule

VAR_INPUT // input vars
	StoredPositions: REFERENCE TO ARRAY[GVL.POS_ARR_BEG..GVL.POS_ARR_END] OF DUT_StoredPosition;
	VisionRegisters: REFERENCE TO ARRAY[GVL.VIS_ARR_BEG..GVL.VIS_ARR_END] OF DUT_VisionRegister;
	Flags: REFERENCE TO ARRAY[GVL.FLG_ARR_BEG..GVL.FLG_ARR_END] OF DUT_Flags;
END_VAR

VAR_OUTPUT // output vars
	ItfUnitMode: PACK_ML.IUnitMode;
	Busy: BOOL;
	Error: BOOL;
	ErrorDescription: STRING;
END_VAR

VAR // standard local vars
	_TimeoutTimer: TON:=(PT:=T#0MS);
	_Home, _Start: BOOL;
	_ModuleFirstScan: BOOL:=TRUE;
	_SeqStart, _SeqHome: INT;
	_AbortedRtrig: R_Trig;
END_VAR

VAR CONSTANT //
	STEP_IDLE: INT := 0000;
	STEP_DONE: INT := 0020;
	STEP_RUN:  INT := 0030;
END_VAR

                    SUPER^();

//
IF _ModuleFirstScan THEN
	ItfUnitMode := SUPER^.IUnitMode;
END_IF;

//
_M_Home();
_M_Start();

//
Busy := _UnitMode.CurrentState <> PACK_ML.State.Idle
		AND _UnitMode.CurrentState <> PACK_ML.State.Aborted
		AND _UnitMode.CurrentState <> PACK_ML.State.Complete
		AND _UnitMode.CurrentState <> PACK_ML.State.Held
		AND _UnitMode.CurrentState <> PACK_ML.State.Stopped
		AND _UnitMode.CurrentState <> PACK_ML.State.Suspended;
		
//
_AbortedRtrig(CLK:=_UnitMode.CurrentState = PACK_ML.State.Aborted);
IF _AbortedRtrig.Q THEN
	//_SeqStart := 0;  _Start:=FALSE;
	//_SeqHome := 0; _Home:=FALSE;
END_IF

//
_TimeoutTimer(IN:= Busy AND _TimeoutTimer.PT > T#0MS); // ignore if timer set to 0
IF _TimeoutTimer.Q THEN
	M_Error(Description:= CONCAT('Task timed out after ', TIME_TO_STRING(_TimeoutTimer.ET)));
END_IF

// do not place anything below this
_ModuleFirstScan:=FALSE;
                  

METHOD PUBLIC M_Start
VAR_INPUT
END_VAR
                          _Start := TRUE;
                        
END_METHOD

METHOD PUBLIC M_Home
VAR_INPUT
END_VAR
                          _Home:=TRUE;
                        
END_METHOD

METHOD PROTECTED M_Error : BOOL
VAR_INPUT
	Description: STRING;
END_VAR
                          // suspend state machine
_UnitMode.Suspend();

//
Error := TRUE;

//
IF ErrorDescription = '' THEN
	ErrorDescription := Description;
ELSE // add a space and tack on the additional error description
	ErrorDescription := CONCAT(ErrorDescription, ' ');
	ErrorDescription := CONCAT(ErrorDescription, Description);
END_IF

GVL.sLastFault := ErrorDescription;
AlarmManager.AlarmGlobals.g_AlarmHandler.RaiseEvent(
    Alm_AlarmConfiguration_Alarmgroup_IDs.ID_Processors,
    Alm_Processors_Alarm_IDs.ID_ProcessorFault);
                        
END_METHOD

METHOD PUBLIC M_Abort
VAR_INPUT
END_VAR
                          _UnitMode.Abort();
_SeqStart := 0;  _Start:=FALSE;
_SeqHome := 0; _Home:=FALSE;
                        
END_METHOD

METHOD PUBLIC M_Hold
VAR_INPUT
END_VAR
                          _UnitMode.Hold();
                        
END_METHOD

METHOD PUBLIC M_Stop
VAR_INPUT
END_VAR
                          _UnitMode.Stop();
                        
END_METHOD

METHOD PRIVATE _M_Start : BOOL
                          CASE _SeqStart OF
	0:
		IF _Start THEN
			_Start := FALSE;
			M_Reset();
			_SeqStart := _SeqStart + 1;
		END_IF
	1:
		CASE _UnitMode.CurrentState OF
			PACK_ML.State.Clearing,
			PACK_ML.State.Resetting,
			PACK_ML.State.UnHolding,
			PACK_ML.State.UnSuspending,
			PACK_ML.State.Starting:
				// be patient
			PACK_ML.State.Aborted:
				_UnitMode.Clear();
			PACK_ML.State.Stopped:
				_UnitMode.Reset();
			PACK_ML.State.Held:
				_UnitMode.UnHold();
			PACK_ML.State.Suspended:
				_UnitMode.UnSuspend();
			PACK_ML.State.Idle:
				_UnitMode.Start();
			PACK_ML.State.Execute:
				_SeqStart := 0;
		ELSE
			_SeqStart := 0;
		END_CASE
		
END_CASE
                        
END_METHOD

METHOD PROTECTED M_Reset : BOOL
VAR_INPUT
END_VAR
                          Error := FALSE;
ErrorDescription := '';
                        
END_METHOD

METHOD PRIVATE _M_Home : BOOL
                          CASE _SeqHome OF
	0:
		//
		IF _Home THEN
			_Home := FALSE;
			M_Reset();
			_SeqHome := _SeqHome + 1;
		END_IF
	1:
		//
		CASE _UnitMode.CurrentState OF
			PACK_ML.State.Aborted:
				_UnitMode.Clear();
				
			PACK_ML.State.Stopped,
			PACK_ML.State.Complete:
				_UnitMode.Reset();
				_SeqHome := _SeqHome + 1;
				
			PACK_ML.State.Resetting,
			PACK_ML.State.Clearing,
			PACK_ML.State.Aborting:
				// just wait
		ELSE
			_UnitMode.Abort();
			
		END_CASE
		
	2:
		IF _UnitMode.CurrentState = PACK_ML.State.Idle THEN
			_SeqHome := 0;
		END_IF
		
END_CASE
                        
END_METHOD

{attribute 'monitoring' := 'variable'}
PROPERTY PropCurrentState : PACK_ML.State
GET
VAR
END_VAR
                            PropCurrentState := ItfUnitMode.CurrentState;
                          
END_GET
END_PROPERTY

{attribute 'monitoring' := 'variable'}
PROPERTY PropBusy : BOOL
GET
VAR
END_VAR
                            PropBusy := Busy;
                          
END_GET
END_PROPERTY

{attribute 'monitoring' := 'variable'}
PROPERTY PropError : BOOL
GET
VAR
END_VAR
                            PropError := Error;
                          
END_GET
END_PROPERTY

{attribute 'monitoring' := 'variable'}
PROPERTY PropErrDescription : STRING
GET
VAR
END_VAR
                            PropErrDescription := ErrorDescription;
                          
END_GET
END_PROPERTY
END_FUNCTION_BLOCK

FUNCTION_BLOCK FB_VisionCmdProcessor EXTENDS FB_Module
VAR_INPUT
	Command: STRING(GVL.COMMAND_LEN):='';
	LogicCmdIO: REFERENCE TO ST_LogicCmdIO;
	VisionSystemIpAddress: STRING(19):='127.0.0.1';
	VisionSystemPort: UINT:=50011;
END_VAR
VAR_OUTPUT
	VisionStateText: STRING:='READY';
END_VAR
VAR
	_CaptureImage_Output: STRING(255);
	_CaptureImage_WorkerUid: STRING;
	_LocatePart_Output: STRING(255);
	_LocatePart_WorkerUid: STRING;
	_RunCalibration_Output: STRING(255);
	_RunCalibration_WorkerUid: STRING;
    _Vision: FB_OpenCV;
    _VisionCommandParser: FB_ParseVisionCmd;
    _VisionDoneRtrig: R_TRIG;
	_VisionBusyRtrig: R_TRIG;
	_VisionResult: STRING(255);
	_ResultPosition: INT;
	_ResultPosition_CAL: INT;
	_ResultPosition_LOC: INT;
	_ResultPosition_CAP: INT;
	_SpacePosition: INT;
	_VisionObjectIndex: UINT;
	_VisionRatio: REAL;
	_VisionRotation: REAL;
	_VisionError: REAL;
	_PartsCount: UDINT;
	_UnitModeCurrentState: PACK_ML.State;
END_VAR

VAR CONSTANT
	_RESPONSE_CAL:          STRING:='res: CAL ';
	_RESPONSE_LOC:          STRING:='res: LOC ';
	_RESPONSE_CAP:          STRING:='res: CAP ';

	_STEP_DONE: 			INT := 1000;
	_STEP_IDLE: 			INT := 0000;
	_STEP_COMMAND: 			INT := 0020;
	_STEP_TRIGGER: 			INT := 0030;
	_STEP_WAIT: 			INT := 0040;
	_STEP_ERR: 				INT := 0050;
END_VAR

                    SUPER^();

// PackML state machine implementation
_UnitModeCurrentState := SUPER^._UnitMode.CurrentState;

//
CASE SUPER^._SeqMain OF
	
    _STEP_DONE:
		SUPER^._SeqMain := _STEP_IDLE;
        
    _STEP_IDLE:
		// hang out here until called to run
        
    _STEP_COMMAND: // parse vision command
        _VisionCommandParser(Command:=Command);
		IF _VisionCommandParser.Error THEN
			SUPER^.M_Error(Description:=_VisionCommandParser.ErrorDescription);
			//
			SUPER^._SeqMain := _STEP_ERR;
		ELSE
			IF _VisionCommandParser.stCommand.Timeout > 0 THEN
				SUPER^._TimeoutTimer.PT := UDINT_TO_TIME(_VisionCommandParser.stCommand.Timeout * 1000);
			END_IF
			//
			SUPER^._SeqMain := _STEP_TRIGGER;
		END_IF
		
	_STEP_TRIGGER: //
		CASE _VisionCommandParser.stCommand.CommandType OF
			DUT_Command_VisionType.Calibrate: //
				_Vision.M_CalibrateCamera(	iImageWidth:= _VisionCommandParser.stCommand.ImageWidth, 
											iImageHeight:= _VisionCommandParser.stCommand.ImageHeight, 
											fCalCheckerSize:= _VisionCommandParser.stCommand.Calibrate.CheckerSize, 
											iCalCheckerX:= _VisionCommandParser.stCommand.Calibrate.CheckerXCount, 
											iCalCheckerY:= _VisionCommandParser.stCommand.Calibrate.CheckerYCount,
                                            uTimeout:=_VisionCommandParser.stCommand.Timeout);
			
			DUT_Command_VisionType.Capture: //
				_Vision.M_CaptureImage(	iImageWidth:= _VisionCommandParser.stCommand.ImageWidth, 
										iImageHeight:= _VisionCommandParser.stCommand.ImageHeight,
                                        uTimeout:=_VisionCommandParser.stCommand.Timeout);
			
			DUT_Command_VisionType.LocatePart: //
                // clear the parts count register
				_PartsCount := 0;
				LogicCmdIO.Register[_VisionCommandParser.stCommand.Locate.ResultPosition] := 0;
                
                // call vision
				_Vision.M_LocatePart( 	iImageWidth:= _VisionCommandParser.stCommand.ImageWidth, 
										iImageHeight:= _VisionCommandParser.stCommand.ImageHeight, 
										iMaxPos:= _VisionCommandParser.stCommand.Locate.MaxParts, 
										dMaxOverlap:= _VisionCommandParser.stCommand.Locate.MaxOverlap, 
										dScore:= _VisionCommandParser.stCommand.Locate.Score, 
										dToleranceAngle:= _VisionCommandParser.stCommand.Locate.ToleranceAngle,
                                        uTimeout:=_VisionCommandParser.stCommand.Timeout,
										sTemplateName:=_VisionCommandParser.stCommand.Locate.TemplateName,
										sScriptFilename:=_VisionCommandParser.stCommand.Locate.ScriptFilename);
			
		END_CASE;
		
		//
		SUPER^._SeqMain := _STEP_WAIT;
		
	_STEP_WAIT: //
		IF _VisionDoneRtrig.Q THEN
			
			//
			_VisionResult := _Vision.P_Response;
			
			//
			_ResultPosition_CAL := FIND(STR1:=_VisionResult,STR2:=_RESPONSE_CAL);
			_ResultPosition_LOC := FIND(STR1:=_VisionResult,STR2:=_RESPONSE_LOC);
			_ResultPosition_CAP := FIND(STR1:=_VisionResult,STR2:=_RESPONSE_CAP);
			
